  LIN {X -16169.500,Y -1557.401,Z 8.000,A 90.00000,B 0.00000,C 180.00000} ; retreat
  ; Step 222, bar 3419
  LIN {X 16169.500,Y -1557.401,Z 792.630,A 90.00000,B 0.00000,C 180.00000} ; outside
  LIN {X 16169.500,Y -1557.401,Z -42.000,A 90.00000,B 0.00000,C 180.00000} ; preinsert
  LIN {X 16169.500,Y -1557.401,Z -292.000,A 90.00000,B 0.00000,C 180.00000} ; insert
  LIN {X 16169.500,Y -1557.401,Z -292.000,A 90.00000,B 0.00000,C 180.00000} ; release
  LIN {X 16169.500,Y -1557.401,Z 8.000,A 90.00000,B 0.00000,C 180.00000} ; retreat
  ; Step 223, bar 3421
  LIN {X -16169.500,Y 1557.401,Z 792.630,A -90.00000,B 0.00000,C 180.00000} ; outside
  LIN {X -16169.500,Y 1557.401,Z -42.000,A -90.00000,B 0.00000,C 180.00000} ; preinsert
  LIN {X -16169.500,Y 1557.401,Z -292.000,A -90.00000,B 0.00000,C 180.00000} ; insert
  LIN {X -16169.500,Y 1557.401,Z -292.000,A -90.00000,B 0.00000,C 180.00000} ; release
  LIN {X -16169.500,Y 1557.401,Z 8.000,A -90.00000,B 0.00000,C 180.00000} ; retreat
  ; Step 224, bar 3417
  LIN {X 16169.500,Y 1557.401,Z 792.630,A -90.00000,B 0.00000,C 180.00000} ; outside
  LIN {X 16169.500,Y 1557.401,Z -42.000,A -90.00000,B 0.00000,C 180.00000} ; preinsert
  LIN {X 16169.500,Y 1557.401,Z -292.000,A -90.00000,B 0.00000,C 180.00000} ; insert
  LIN {X 16169.500,Y 1557.401,Z -292.000,A -90.00000,B 0.00000,C 180.00000} ; release
  LIN {X 16169.500,Y 1557.401,Z 8.000,A -90.00000,B 0.00000,C 180.00000} ; retreat
  ; Step 225, bar 1865
  LIN {X 0.000,Y -2739.855,Z 792.630,A 0.00000,B 0.00000,C 180.00000} ; outside
  LIN {X 0.000,Y -2739.855,Z -37.029,A 0.00000,B 0.00000,C 180.00000} ; preinsert
  LIN {X 0.000,Y -2739.855,Z -287.029,A 0.00000,B 0.00000,C 180.00000} ; insert
  LIN {X 0.000,Y -2739.855,Z -287.029,A 0.00000,B 0.00000,C 180.00000} ; release
  LIN {X 0.000,Y -2739.855,Z 12.971,A 0.00000,B 0.00000,C 180.00000} ; retreat
  ; Step 226, bar 1878
  LIN {X 0.000,Y 2739.855,Z 792.630,A 0.00000,B 0.00000,C 180.00000} ; outside
  LIN {X 0.000,Y 2739.855,Z -37.029,A 0.00000,B 0.00000,C 180.00000} ; preinsert
  LIN {X 0.000,Y 2739.855,Z -287.029,A 0.00000,B 0.00000,C 180.00000} ; insert
  LIN {X 0.000,Y 2739.855,Z -287.029,A 0.00000,B 0.00000,C 180.00000} ; release
  LIN {X 0.000,Y 2739.855,Z 12.971,A 0.00000,B 0.00000,C 180.00000} ; retreat
  ; Step 227, bar 1060
  LIN {X 16149.984,Y 0.199,Z 793.369,A 90.00387,B 0.00000,C 180.00000} ; outside
  LIN {X 16149.984,Y 0.199,Z -166.684,A 90.00387,B 0.00000,C 180.00000} ; preinsert
  LIN {X 16149.984,Y 0.199,Z -416.684,A 90.00387,B 0.00000,C 180.00000} ; insert
  LIN {X 16149.984,Y 0.199,Z -416.684,A 90.00387,B 0.00000,C 180.00000} ; release
  LIN {X 16149.984,Y 0.199,Z -116.684,A 90.00387,B 0.00000,C 180.00000} ; retreat
  ; Step 228, bar 1061
  LIN {X 16249.984,Y 0.199,Z 793.369,A 90.00387,B 0.00000,C 180.00000} ; outside
  LIN {X 16249.984,Y 0.199,Z -166.684,A 90.00387,B 0.00000,C 180.00000} ; preinsert
  LIN {X 16249.984,Y 0.199,Z -416.684,A 90.00387,B 0.00000,C 180.00000} ; insert
  LIN {X 16249.984,Y 0.199,Z -416.684,A 90.00387,B 0.00000,C 180.00000} ; release
  LIN {X 16249.984,Y 0.199,Z -116.684,A 90.00387,B 0.00000,C 180.00000} ; retreat
  ; Step 229, bar 1847
  LIN {X -16149.984,Y 0.199,Z 793.369,A 89.99613,B 0.00000,C -180.00000} ; outside
  LIN {X -16149.984,Y 0.199,Z -166.684,A 89.99613,B 0.00000,C -180.00000} ; preinsert
  LIN {X -16149.984,Y 0.199,Z -416.684,A 89.99613,B 0.00000,C -180.00000} ; insert
  LIN {X -16149.984,Y 0.199,Z -416.684,A 89.99613,B 0.00000,C -180.00000} ; release
  LIN {X -16149.984,Y 0.199,Z -116.684,A 89.99613,B 0.00000,C -180.00000} ; retreat
  ; Step 230, bar 1848
  LIN {X -16249.984,Y 0.199,Z 793.369,A 89.99613,B 0.00000,C -180.00000} ; outside
  LIN {X -16249.984,Y 0.199,Z -166.684,A 89.99613,B 0.00000,C -180.00000} ; preinsert
  LIN {X -16249.984,Y 0.199,Z -416.684,A 89.99613,B 0.00000,C -180.00000} ; insert
  LIN {X -16249.984,Y 0.199,Z -416.684,A 89.99613,B 0.00000,C -180.00000} ; release
  LIN {X -16249.984,Y 0.199,Z -116.684,A 89.99613,B 0.00000,C -180.00000} ; retreat
  ; Step 231, bar 1051
  LIN {X 15249.971,Y 0.435,Z 793.207,A 89.99774,B 0.00000,C 180.00000} ; outside
  LIN {X 15249.971,Y 0.435,Z -166.823,A 89.99774,B 0.00000,C 180.00000} ; preinsert
  LIN {X 15249.971,Y 0.435,Z -416.823,A 89.99774,B 0.00000,C 180.00000} ; insert
  LIN {X 15249.971,Y 0.435,Z -416.823,A 89.99774,B 0.00000,C 180.00000} ; release
  LIN {X 15249.971,Y 0.435,Z -116.823,A 89.99774,B 0.00000,C 180.00000} ; retreat
  ; Step 232, bar 1052
  LIN {X 15349.971,Y 0.435,Z 793.207,A 89.99774,B 0.00000,C 180.00000} ; outside
  LIN {X 15349.971,Y 0.435,Z -166.823,A 89.99774,B 0.00000,C 180.00000} ; preinsert
  LIN {X 15349.971,Y 0.435,Z -416.823,A 89.99774,B 0.00000,C 180.00000} ; insert
  LIN {X 15349.971,Y 0.435,Z -416.823,A 89.99774,B 0.00000,C 180.00000} ; release
  LIN {X 15349.971,Y 0.435,Z -116.823,A 89.99774,B 0.00000,C 180.00000} ; retreat
  ; Step 233, bar 1053
  LIN {X 15449.971,Y 0.435,Z 793.207,A 89.99774,B 0.00000,C 180.00000} ; outside
  LIN {X 15449.971,Y 0.435,Z -166.823,A 89.99774,B 0.00000,C 180.00000} ; preinsert
  LIN {X 15449.971,Y 0.435,Z -416.823,A 89.99774,B 0.00000,C 180.00000} ; insert
  LIN {X 15449.971,Y 0.435,Z -416.823,A 89.99774,B 0.00000,C 180.00000} ; release
  LIN {X 15449.971,Y 0.435,Z -116.823,A 89.99774,B 0.00000,C 180.00000} ; retreat
  ; Step 234, bar 1055
  LIN {X 15649.971,Y 0.435,Z 793.207,A 89.99774,B 0.00000,C 180.00000} ; outside
  LIN {X 15649.971,Y 0.435,Z -166.823,A 89.99774,B 0.00000,C 180.00000} ; preinsert
  LIN {X 15649.971,Y 0.435,Z -416.823,A 89.99774,B 0.00000,C 180.00000} ; insert
  LIN {X 15649.971,Y 0.435,Z -416.823,A 89.99774,B 0.00000,C 180.00000} ; release
  LIN {X 15649.971,Y 0.435,Z -116.823,A 89.99774,B 0.00000,C 180.00000} ; retreat
  ; Step 235, bar 1056
  LIN {X 15749.971,Y 0.435,Z 793.207,A 89.99774,B 0.00000,C 180.00000} ; outside
  LIN {X 15749.971,Y 0.435,Z -166.823,A 89.99774,B 0.00000,C 180.00000} ; preinsert
  LIN {X 15749.971,Y 0.435,Z -416.823,A 89.99774,B 0.00000,C 180.00000} ; insert
  LIN {X 15749.971,Y 0.435,Z -416.823,A 89.99774,B 0.00000,C 180.00000} ; release
  LIN {X 15749.971,Y 0.435,Z -116.823,A 89.99774,B 0.00000,C 180.00000} ; retreat
  ; Step 236, bar 1057
  LIN {X 15849.971,Y 0.435,Z 793.207,A 89.99774,B 0.00000,C 180.00000} ; outside
  LIN {X 15849.971,Y 0.435,Z -166.823,A 89.99774,B 0.00000,C 180.00000} ; preinsert
  LIN {X 15849.971,Y 0.435,Z -416.823,A 89.99774,B 0.00000,C 180.00000} ; insert
  LIN {X 15849.971,Y 0.435,Z -416.823,A 89.99774,B 0.00000,C 180.00000} ; release
  LIN {X 15849.971,Y 0.435,Z -116.823,A 89.99774,B 0.00000,C 180.00000} ; retreat
  ; Step 237, bar 1058
  LIN {X 15949.971,Y 0.435,Z 793.207,A 89.99774,B 0.00000,C 180.00000} ; outside
  LIN {X 15949.971,Y 0.435,Z -166.823,A 89.99774,B 0.00000,C 180.00000} ; preinsert
  LIN {X 15949.971,Y 0.435,Z -416.823,A 89.99774,B 0.00000,C 180.00000} ; insert
  LIN {X 15949.971,Y 0.435,Z -416.823,A 89.99774,B 0.00000,C 180.00000} ; release
  LIN {X 15949.971,Y 0.435,Z -116.823,A 89.99774,B 0.00000,C 180.00000} ; retreat
  ; Step 238, bar 1059
  LIN {X 16049.971,Y 0.435,Z 793.207,A 89.99774,B 0.00000,C 180.00000} ; outside
  LIN {X 16049.971,Y 0.435,Z -166.823,A 89.99774,B 0.00000,C 180.00000} ; preinsert
  LIN {X 16049.971,Y 0.435,Z -416.823,A 89.99774,B 0.00000,C 180.00000} ; insert
  LIN {X 16049.971,Y 0.435,Z -416.823,A 89.99774,B 0.00000,C 180.00000} ; release
  LIN {X 16049.971,Y 0.435,Z -116.823,A 89.99774,B 0.00000,C 180.00000} ; retreat
  ; Step 239, bar 1799
  LIN {X -15249.971,Y 0.435,Z 793.207,A 90.00226,B 0.00000,C 180.00000} ; outside
  LIN {X -15249.971,Y 0.435,Z -166.823,A 90.00226,B 0.00000,C 180.00000} ; preinsert
  LIN {X -15249.971,Y 0.435,Z -416.823,A 90.00226,B 0.00000,C 180.00000} ; insert
  LIN {X -15249.971,Y 0.435,Z -416.823,A 90.00226,B 0.00000,C 180.00000} ; release
  LIN {X -15249.971,Y 0.435,Z -116.823,A 90.00226,B 0.00000,C 180.00000} ; retreat
  ; Step 240, bar 1800
  LIN {X -15349.971,Y 0.435,Z 793.207,A 90.00226,B 0.00000,C 180.00000} ; outside
  LIN {X -15349.971,Y 0.435,Z -166.823,A 90.00226,B 0.00000,C 180.00000} ; preinsert
  LIN {X -15349.971,Y 0.435,Z -416.823,A 90.00226,B 0.00000,C 180.00000} ; insert
  LIN {X -15349.971,Y 0.435,Z -416.823,A 90.00226,B 0.00000,C 180.00000} ; release
  LIN {X -15349.971,Y 0.435,Z -116.823,A 90.00226,B 0.00000,C 180.00000} ; retreat
  ; Step 241, bar 1801
  LIN {X -15449.971,Y 0.435,Z 793.207,A 90.00226,B 0.00000,C 180.00000} ; outside
  LIN {X -15449.971,Y 0.435,Z -166.823,A 90.00226,B 0.00000,C 180.00000} ; preinsert
  LIN {X -15449.971,Y 0.435,Z -416.823,A 90.00226,B 0.00000,C 180.00000} ; insert
  LIN {X -15449.971,Y 0.435,Z -416.823,A 90.00226,B 0.00000,C 180.00000} ; release
  LIN {X -15449.971,Y 0.435,Z -116.823,A 90.00226,B 0.00000,C 180.00000} ; retreat
  ; Step 242, bar 1802
  LIN {X -15649.971,Y 0.435,Z 793.207,A 90.00226,B 0.00000,C 180.00000} ; outside
  LIN {X -15649.971,Y 0.435,Z -166.823,A 90.00226,B 0.00000,C 180.00000} ; preinsert
  LIN {X -15649.971,Y 0.435,Z -416.823,A 90.00226,B 0.00000,C 180.00000} ; insert
  LIN {X -15649.971,Y 0.435,Z -416.823,A 90.00226,B 0.00000,C 180.00000} ; release
  LIN {X -15649.971,Y 0.435,Z -116.823,A 90.00226,B 0.00000,C 180.00000} ; retreat
  ; Step 243, bar 1803
  LIN {X -15749.971,Y 0.435,Z 793.207,A 90.00226,B 0.00000,C 180.00000} ; outside
  LIN {X -15749.971,Y 0.435,Z -166.823,A 90.00226,B 0.00000,C 180.00000} ; preinsert
  LIN {X -15749.971,Y 0.435,Z -416.823,A 90.00226,B 0.00000,C 180.00000} ; insert
  LIN {X -15749.971,Y 0.435,Z -416.823,A 90.00226,B 0.00000,C 180.00000} ; release
  LIN {X -15749.971,Y 0.435,Z -116.823,A 90.00226,B 0.00000,C 180.00000} ; retreat
  ; Step 244, bar 1804
  LIN {X -15849.971,Y 0.435,Z 793.207,A 90.00226,B 0.00000,C 180.00000} ; outside
  LIN {X -15849.971,Y 0.435,Z -166.823,A 90.00226,B 0.00000,C 180.00000} ; preinsert
  LIN {X -15849.971,Y 0.435,Z -416.823,A 90.00226,B 0.00000,C 180.00000} ; insert
  LIN {X -15849.971,Y 0.435,Z -416.823,A 90.00226,B 0.00000,C 180.00000} ; release
  LIN {X -15849.971,Y 0.435,Z -116.823,A 90.00226,B 0.00000,C 180.00000} ; retreat
  ; Step 245, bar 1805
  LIN {X -15949.971,Y 0.435,Z 793.207,A 90.00226,B 0.00000,C 180.00000} ; outside
  LIN {X -15949.971,Y 0.435,Z -166.823,A 90.00226,B 0.00000,C 180.00000} ; preinsert
  LIN {X -15949.971,Y 0.435,Z -416.823,A 90.00226,B 0.00000,C 180.00000} ; insert
  LIN {X -15949.971,Y 0.435,Z -416.823,A 90.00226,B 0.00000,C 180.00000} ; release
  LIN {X -15949.971,Y 0.435,Z -116.823,A 90.00226,B 0.00000,C 180.00000} ; retreat
  ; Step 246, bar 1806
  LIN {X -16049.971,Y 0.435,Z 793.207,A 90.00226,B 0.00000,C 180.00000} ; outside
  LIN {X -16049.971,Y 0.435,Z -166.823,A 90.00226,B 0.00000,C 180.00000} ; preinsert
  LIN {X -16049.971,Y 0.435,Z -416.823,A 90.00226,B 0.00000,C 180.00000} ; insert
  LIN {X -16049.971,Y 0.435,Z -416.823,A 90.00226,B 0.00000,C 180.00000} ; release
  LIN {X -16049.971,Y 0.435,Z -116.823,A 90.00226,B 0.00000,C 180.00000} ; retreat
  ; Step 247, bar 1866
  LIN {X 0.000,Y -2889.855,Z 792.630,A 0.00000,B 0.00000,C 180.00000} ; outside
  LIN {X 0.000,Y -2889.855,Z -19.788,A 0.00000,B 0.00000,C 180.00000} ; preinsert
  LIN {X 0.000,Y -2889.855,Z -269.788,A 0.00000,B 0.00000,C 180.00000} ; insert
  LIN {X 0.000,Y -2889.855,Z -269.788,A 0.00000,B 0.00000,C 180.00000} ; release
  LIN {X 0.000,Y -2889.855,Z 30.212,A 0.00000,B 0.00000,C 180.00000} ; retreat
  ; Step 248, bar 1879
  LIN {X 0.000,Y 2889.855,Z 792.630,A 0.00000,B 0.00000,C 180.00000} ; outside
  LIN {X 0.000,Y 2889.855,Z -19.788,A 0.00000,B 0.00000,C 180.00000} ; preinsert
  LIN {X 0.000,Y 2889.855,Z -269.788,A 0.00000,B 0.00000,C 180.00000} ; insert
  LIN {X 0.000,Y 2889.855,Z -269.788,A 0.00000,B 0.00000,C 180.00000} ; release
  LIN {X 0.000,Y 2889.855,Z 30.212,A 0.00000,B 0.00000,C 180.00000} ; retreat
  ; Step 249, bar 1050
  LIN {X 15149.971,Y 0.435,Z 793.207,A 89.99774,B 0.00000,C 180.00000} ; outside
  LIN {X 15149.971,Y 0.435,Z -163.267,A 89.99774,B 0.00000,C 180.00000} ; preinsert
  LIN {X 15149.971,Y 0.435,Z -413.267,A 89.99774,B 0.00000,C 180.00000} ; insert
  LIN {X 15149.971,Y 0.435,Z -413.267,A 89.99774,B 0.00000,C 180.00000} ; release
  LIN {X 15149.971,Y 0.435,Z -113.267,A 89.99774,B 0.00000,C 180.00000} ; retreat
  ; Step 250, bar 1798
  LIN {X -15149.971,Y 0.435,Z 793.207,A 90.00226,B 0.00000,C 180.00000} ; outside
  LIN {X -15149.971,Y 0.435,Z -163.267,A 90.00226,B 0.00000,C 180.00000} ; preinsert
  LIN {X -15149.971,Y 0.435,Z -413.267,A 90.00226,B 0.00000,C 180.00000} ; insert
  LIN {X -15149.971,Y 0.435,Z -413.267,A 90.00226,B 0.00000,C 180.00000} ; release
  LIN {X -15149.971,Y 0.435,Z -113.267,A 90.00226,B 0.00000,C 180.00000} ; retreat
  ; Step 251, bar 1049
  LIN {X 15049.971,Y 0.435,Z 793.207,A 89.99774,B 0.00000,C 180.00000} ; outside
  LIN {X 15049.971,Y 0.435,Z -156.587,A 89.99774,B 0.00000,C 180.00000} ; preinsert
  LIN {X 15049.971,Y 0.435,Z -406.587,A 89.99774,B 0.00000,C 180.00000} ; insert
  LIN {X 15049.971,Y 0.435,Z -406.587,A 89.99774,B 0.00000,C 180.00000} ; release
  LIN {X 15049.971,Y 0.435,Z -106.587,A 89.99774,B 0.00000,C 180.00000} ; retreat
  ; Step 252, bar 1797
  LIN {X -15049.971,Y 0.435,Z 793.207,A 90.00226,B 0.00000,C 180.00000} ; outside
  LIN {X -15049.971,Y 0.435,Z -156.587,A 90.00226,B 0.00000,C 180.00000} ; preinsert
  LIN {X -15049.971,Y 0.435,Z -406.587,A 90.00226,B 0.00000,C 180.00000} ; insert
  LIN {X -15049.971,Y 0.435,Z -406.587,A 90.00226,B 0.00000,C 180.00000} ; release
  LIN {X -15049.971,Y 0.435,Z -106.587,A 90.00226,B 0.00000,C 180.00000} ; retreat
  ; Step 253, bar 1048
  LIN {X 14949.971,Y 0.435,Z 793.207,A 89.99774,B 0.00000,C 180.00000} ; outside
  LIN {X 14949.971,Y 0.435,Z -149.906,A 89.99774,B 0.00000,C 180.00000} ; preinsert
  LIN {X 14949.971,Y 0.435,Z -399.906,A 89.99774,B 0.00000,C 180.00000} ; insert
  LIN {X 14949.971,Y 0.435,Z -399.906,A 89.99774,B 0.00000,C 180.00000} ; release
  LIN {X 14949.971,Y 0.435,Z -99.906,A 89.99774,B 0.00000,C 180.00000} ; retreat
  ; Step 254, bar 1796
  LIN {X -14949.971,Y 0.435,Z 793.207,A 90.00226,B 0.00000,C 180.00000} ; outside
  LIN {X -14949.971,Y 0.435,Z -149.906,A 90.00226,B 0.00000,C 180.00000} ; preinsert
  LIN {X -14949.971,Y 0.435,Z -399.906,A 90.00226,B 0.00000,C 180.00000} ; insert
  LIN {X -14949.971,Y 0.435,Z -399.906,A 90.00226,B 0.00000,C 180.00000} ; release
  LIN {X -14949.971,Y 0.435,Z -99.906,A 90.00226,B 0.00000,C 180.00000} ; retreat
  ; Step 255, bar 1950
  LIN {X 0.000,Y -1050.000,Z 792.630,A 0.00000,B 0.00000,C 180.00000} ; outside
  LIN {X 0.000,Y -1050.000,Z -2.875,A 0.00000,B 0.00000,C 180.00000} ; preinsert
  LIN {X 0.000,Y -1050.000,Z -252.875,A 0.00000,B 0.00000,C 180.00000} ; insert
  LIN {X 0.000,Y -1050.000,Z -252.875,A 0.00000,B 0.00000,C 180.00000} ; release
  LIN {X 0.000,Y -1050.000,Z 47.125,A 0.00000,B 0.00000,C 180.00000} ; retreat
  ; Step 256, bar 1945
  LIN {X 0.000,Y 1050.000,Z 792.630,A 0.00000,B 0.00000,C 180.00000} ; outside
  LIN {X 0.000,Y 1050.000,Z -2.875,A 0.00000,B 0.00000,C 180.00000} ; preinsert
  LIN {X 0.000,Y 1050.000,Z -252.875,A 0.00000,B 0.00000,C 180.00000} ; insert
  LIN {X 0.000,Y 1050.000,Z -252.875,A 0.00000,B 0.00000,C 180.00000} ; release
  LIN {X 0.000,Y 1050.000,Z 47.125,A 0.00000,B 0.00000,C 180.00000} ; retreat
  ; Step 257, bar 1867
  LIN {X 0.000,Y -3039.855,Z 792.630,A 0.00000,B 0.00000,C 180.00000} ; outside
  LIN {X 0.000,Y -3039.855,Z -2.546,A 0.00000,B 0.00000,C 180.00000} ; preinsert
  LIN {X 0.000,Y -3039.855,Z -252.546,A 0.00000,B 0.00000,C 180.00000} ; insert
  LIN {X 0.000,Y -3039.855,Z -252.546,A 0.00000,B 0.00000,C 180.00000} ; release
  LIN {X 0.000,Y -3039.855,Z 47.454,A 0.00000,B 0.00000,C 180.00000} ; retreat
  ; Step 258, bar 1880
  LIN {X 0.000,Y 3039.855,Z 792.630,A 0.00000,B 0.00000,C 180.00000} ; outside
  LIN {X 0.000,Y 3039.855,Z -2.546,A 0.00000,B 0.00000,C 180.00000} ; preinsert
  LIN {X 0.000,Y 3039.855,Z -252.546,A 0.00000,B 0.00000,C 180.00000} ; insert
  LIN {X 0.000,Y 3039.855,Z -252.546,A 0.00000,B 0.00000,C 180.00000} ; release
  LIN {X 0.000,Y 3039.855,Z 47.454,A 0.00000,B 0.00000,C 180.00000} ; retreat
  ; Step 259, bar 1047
  LIN {X 14849.971,Y 0.435,Z 793.207,A 89.99774,B 0.00000,C 180.00000} ; outside
  LIN {X 14849.971,Y 0.435,Z -143.225,A 89.99774,B 0.00000,C 180.00000} ; preinsert
  LIN {X 14849.971,Y 0.435,Z -393.225,A 89.99774,B 0.00000,C 180.00000} ; insert
  LIN {X 14849.971,Y 0.435,Z -393.225,A 89.99774,B 0.00000,C 180.00000} ; release
  LIN {X 14849.971,Y 0.435,Z -93.225,A 89.99774,B 0.00000,C 180.00000} ; retreat
  ; Step 260, bar 1795
  LIN {X -14849.971,Y 0.435,Z 793.207,A 90.00226,B 0.00000,C 180.00000} ; outside
  LIN {X -14849.971,Y 0.435,Z -143.225,A 90.00226,B 0.00000,C 180.00000} ; preinsert
  LIN {X -14849.971,Y 0.435,Z -393.225,A 90.00226,B 0.00000,C 180.00000} ; insert
  LIN {X -14849.971,Y 0.435,Z -393.225,A 90.00226,B 0.00000,C 180.00000} ; release
  LIN {X -14849.971,Y 0.435,Z -93.225,A 90.00226,B 0.00000,C 180.00000} ; retreat
  ; Step 261, bar 1046
  LIN {X 14749.971,Y 0.435,Z 793.207,A 89.99774,B 0.00000,C 180.00000} ; outside
  LIN {X 14749.971,Y 0.435,Z -136.544,A 89.99774,B 0.00000,C 180.00000} ; preinsert
  LIN {X 14749.971,Y 0.435,Z -386.544,A 89.99774,B 0.00000,C 180.00000} ; insert
  LIN {X 14749.971,Y 0.435,Z -386.544,A 89.99774,B 0.00000,C 180.00000} ; release
  LIN {X 14749.971,Y 0.435,Z -86.544,A 89.99774,B 0.00000,C 180.00000} ; retreat
  ; Step 262, bar 1794
  LIN {X -14749.971,Y 0.435,Z 793.207,A 90.00226,B 0.00000,C 180.00000} ; outside
  LIN {X -14749.971,Y 0.435,Z -136.544,A 90.00226,B 0.00000,C 180.00000} ; preinsert
  LIN {X -14749.971,Y 0.435,Z -386.544,A 90.00226,B 0.00000,C 180.00000} ; insert
  LIN {X -14749.971,Y 0.435,Z -386.544,A 90.00226,B 0.00000,C 180.00000} ; release
  LIN {X -14749.971,Y 0.435,Z -86.544,A 90.00226,B 0.00000,C 180.00000} ; retreat
  ; Step 263, bar 1868
  LIN {X 0.000,Y -3154.855,Z 792.630,A 0.00000,B 0.00000,C 180.00000} ; outside
  LIN {X 0.000,Y -3154.855,Z 10.672,A 0.00000,B 0.00000,C 180.00000} ; preinsert
  LIN {X 0.000,Y -3154.855,Z -239.328,A 0.00000,B 0.00000,C 180.00000} ; insert
  LIN {X 0.000,Y -3154.855,Z -239.328,A 0.00000,B 0.00000,C 180.00000} ; release
  LIN {X 0.000,Y -3154.855,Z 60.672,A 0.00000,B 0.00000,C 180.00000} ; retreat
  ; Step 264, bar 1881
  LIN {X 0.000,Y 3154.855,Z 792.630,A 0.00000,B 0.00000,C 180.00000} ; outside
  LIN {X 0.000,Y 3154.855,Z 10.672,A 0.00000,B 0.00000,C 180.00000} ; preinsert
  LIN {X 0.000,Y 3154.855,Z -239.328,A 0.00000,B 0.00000,C 180.00000} ; insert
  LIN {X 0.000,Y 3154.855,Z -239.328,A 0.00000,B 0.00000,C 180.00000} ; release
  LIN {X 0.000,Y 3154.855,Z 60.672,A 0.00000,B 0.00000,C 180.00000} ; retreat
  ; Step 265, bar 1045
  LIN {X 14649.971,Y 0.435,Z 793.207,A 89.99774,B 0.00000,C 180.00000} ; outside
  LIN {X 14649.971,Y 0.435,Z -129.863,A 89.99774,B 0.00000,C 180.00000} ; preinsert
  LIN {X 14649.971,Y 0.435,Z -379.863,A 89.99774,B 0.00000,C 180.00000} ; insert
  LIN {X 14649.971,Y 0.435,Z -379.863,A 89.99774,B 0.00000,C 180.00000} ; release
  LIN {X 14649.971,Y 0.435,Z -79.863,A 89.99774,B 0.00000,C 180.00000} ; retreat
  ; Step 266, bar 1793
  LIN {X -14649.971,Y 0.435,Z 793.207,A 90.00226,B 0.00000,C 180.00000} ; outside
  LIN {X -14649.971,Y 0.435,Z -129.863,A 90.00226,B 0.00000,C 180.00000} ; preinsert
  LIN {X -14649.971,Y 0.435,Z -379.863,A 90.00226,B 0.00000,C 180.00000} ; insert
  LIN {X -14649.971,Y 0.435,Z -379.863,A 90.00226,B 0.00000,C 180.00000} ; release
  LIN {X -14649.971,Y 0.435,Z -79.863,A 90.00226,B 0.00000,C 180.00000} ; retreat
  ; Step 267, bar 1869
  LIN {X 0.000,Y -3264.855,Z 798.011,A 0.00000,B 0.00000,C 180.00000} ; outside
  LIN {X 0.000,Y -3264.855,Z 23.316,A 0.00000,B 0.00000,C 180.00000} ; preinsert
  LIN {X 0.000,Y -3264.855,Z -226.684,A 0.00000,B 0.00000,C 180.00000} ; insert
  LIN {X 0.000,Y -3264.855,Z -226.684,A 0.00000,B 0.00000,C 180.00000} ; release
  LIN {X 0.000,Y -3264.855,Z 73.316,A 0.00000,B 0.00000,C 180.00000} ; retreat
  ; Step 268, bar 1882
  LIN {X 0.000,Y 3264.855,Z 798.011,A 0.00000,B 0.00000,C 180.00000} ; outside
  LIN {X 0.000,Y 3264.855,Z 23.316,A 0.00000,B 0.00000,C 180.00000} ; preinsert
  LIN {X 0.000,Y 3264.855,Z -226.684,A 0.00000,B 0.00000,C 180.00000} ; insert
  LIN {X 0.000,Y 3264.855,Z -226.684,A 0.00000,B 0.00000,C 180.00000} ; release
  LIN {X 0.000,Y 3264.855,Z 73.316,A 0.00000,B 0.00000,C 180.00000} ; retreat
  ; Step 269, bar 1043
  LIN {X 14449.971,Y 0.435,Z 793.207,A 89.99774,B 0.00000,C 180.00000} ; outside
  LIN {X 14449.971,Y 0.435,Z -116.502,A 89.99774,B 0.00000,C 180.00000} ; preinsert
  LIN {X 14449.971,Y 0.435,Z -366.502,A 89.99774,B 0.00000,C 180.00000} ; insert
  LIN {X 14449.971,Y 0.435,Z -366.502,A 89.99774,B 0.00000,C 180.00000} ; release
  LIN {X 14449.971,Y 0.435,Z -66.502,A 89.99774,B 0.00000,C 180.00000} ; retreat
  ; Step 270, bar 1792
  LIN {X -14449.971,Y 0.435,Z 793.207,A 90.00226,B 0.00000,C 180.00000} ; outside
  LIN {X -14449.971,Y 0.435,Z -116.502,A 90.00226,B 0.00000,C 180.00000} ; preinsert
  LIN {X -14449.971,Y 0.435,Z -366.502,A 90.00226,B 0.00000,C 180.00000} ; insert
  LIN {X -14449.971,Y 0.435,Z -366.502,A 90.00226,B 0.00000,C 180.00000} ; release
  LIN {X -14449.971,Y 0.435,Z -66.502,A 90.00226,B 0.00000,C 180.00000} ; retreat
  ; Step 271, bar 1870
  LIN {X 0.000,Y -3354.855,Z 818.700,A 0.00000,B 0.00000,C 180.00000} ; outside
  LIN {X 0.000,Y -3354.855,Z 33.661,A 0.00000,B 0.00000,C 180.00000} ; preinsert
  LIN {X 0.000,Y -3354.855,Z -216.339,A 0.00000,B 0.00000,C 180.00000} ; insert
  LIN {X 0.000,Y -3354.855,Z -216.339,A 0.00000,B 0.00000,C 180.00000} ; release
  LIN {X 0.000,Y -3354.855,Z 83.661,A 0.00000,B 0.00000,C 180.00000} ; retreat
  ; Step 272, bar 1883
  LIN {X 0.000,Y 3354.855,Z 818.700,A 0.00000,B 0.00000,C 180.00000} ; outside
  LIN {X 0.000,Y 3354.855,Z 33.661,A 0.00000,B 0.00000,C 180.00000} ; preinsert
  LIN {X 0.000,Y 3354.855,Z -216.339,A 0.00000,B 0.00000,C 180.00000} ; insert
  LIN {X 0.000,Y 3354.855,Z -216.339,A 0.00000,B 0.00000,C 180.00000} ; release
  LIN {X 0.000,Y 3354.855,Z 83.661,A 0.00000,B 0.00000,C 180.00000} ; retreat
  ; Step 273, bar 1042
  LIN {X 14349.971,Y 0.435,Z 793.207,A 89.99774,B 0.00000,C 180.00000} ; outside
  LIN {X 14349.971,Y 0.435,Z -109.821,A 89.99774,B 0.00000,C 180.00000} ; preinsert
  LIN {X 14349.971,Y 0.435,Z -359.821,A 89.99774,B 0.00000,C 180.00000} ; insert
  LIN {X 14349.971,Y 0.435,Z -359.821,A 89.99774,B 0.00000,C 180.00000} ; release
  LIN {X 14349.971,Y 0.435,Z -59.821,A 89.99774,B 0.00000,C 180.00000} ; retreat
  ; Step 274, bar 1791
  LIN {X -14349.971,Y 0.435,Z 793.207,A 90.00226,B 0.00000,C 180.00000} ; outside
  LIN {X -14349.971,Y 0.435,Z -109.821,A 90.00226,B 0.00000,C 180.00000} ; preinsert
  LIN {X -14349.971,Y 0.435,Z -359.821,A 90.00226,B 0.00000,C 180.00000} ; insert
  LIN {X -14349.971,Y 0.435,Z -359.821,A 90.00226,B 0.00000,C 180.00000} ; release
  LIN {X -14349.971,Y 0.435,Z -59.821,A 90.00226,B 0.00000,C 180.00000} ; retreat
  ; Step 275, bar 1041
  LIN {X 14249.971,Y 0.435,Z 793.207,A 89.99774,B 0.00000,C 180.00000} ; outside
  LIN {X 14249.971,Y 0.435,Z -103.140,A 89.99774,B 0.00000,C 180.00000} ; preinsert
  LIN {X 14249.971,Y 0.435,Z -353.140,A 89.99774,B 0.00000,C 180.00000} ; insert
  LIN {X 14249.971,Y 0.435,Z -353.140,A 89.99774,B 0.00000,C 180.00000} ; release
  LIN {X 14249.971,Y 0.435,Z -53.140,A 89.99774,B 0.00000,C 180.00000} ; retreat
  ; Step 276, bar 1790
  LIN {X -14249.971,Y 0.435,Z 793.207,A 90.00226,B 0.00000,C 180.00000} ; outside
  LIN {X -14249.971,Y 0.435,Z -103.140,A 90.00226,B 0.00000,C 180.00000} ; preinsert
  LIN {X -14249.971,Y 0.435,Z -353.140,A 90.00226,B 0.00000,C 180.00000} ; insert
  LIN {X -14249.971,Y 0.435,Z -353.140,A 90.00226,B 0.00000,C 180.00000} ; release
  LIN {X -14249.971,Y 0.435,Z -53.140,A 90.00226,B 0.00000,C 180.00000} ; retreat
  ; Step 277, bar 1040
  LIN {X 14149.971,Y 0.435,Z 793.207,A 89.99774,B 0.00000,C 180.00000} ; outside
  LIN {X 14149.971,Y 0.435,Z -96.459,A 89.99774,B 0.00000,C 180.00000} ; preinsert
  LIN {X 14149.971,Y 0.435,Z -346.459,A 89.99774,B 0.00000,C 180.00000} ; insert
  LIN {X 14149.971,Y 0.435,Z -346.459,A 89.99774,B 0.00000,C 180.00000} ; release
  LIN {X 14149.971,Y 0.435,Z -46.459,A 89.99774,B 0.00000,C 180.00000} ; retreat
  ; Step 278, bar 1789
  LIN {X -14149.971,Y 0.435,Z 793.207,A 90.00226,B 0.00000,C 180.00000} ; outside
  LIN {X -14149.971,Y 0.435,Z -96.459,A 90.00226,B 0.00000,C 180.00000} ; preinsert
  LIN {X -14149.971,Y 0.435,Z -346.459,A 90.00226,B 0.00000,C 180.00000} ; insert
  LIN {X -14149.971,Y 0.435,Z -346.459,A 90.00226,B 0.00000,C 180.00000} ; release
  LIN {X -14149.971,Y 0.435,Z -46.459,A 90.00226,B 0.00000,C 180.00000} ; retreat
  ; Step 279, bar 1944
  LIN {X 0.000,Y -1420.000,Z 849.379,A 0.00000,B 0.00000,C 180.00000} ; outside
  LIN {X 0.000,Y -1420.000,Z 49.000,A 0.00000,B 0.00000,C 180.00000} ; preinsert
  LIN {X 0.000,Y -1420.000,Z -201.000,A 0.00000,B 0.00000,C 180.00000} ; insert
  LIN {X 0.000,Y -1420.000,Z -201.000,A 0.00000,B 0.00000,C 180.00000} ; release
  LIN {X 0.000,Y -1420.000,Z 99.000,A 0.00000,B 0.00000,C 180.00000} ; retreat
  ; Step 280, bar 1943
  LIN {X 0.000,Y -1050.000,Z 849.379,A 0.00000,B 0.00000,C 180.00000} ; outside
  LIN {X 0.000,Y -1050.000,Z 49.000,A 0.00000,B 0.00000,C 180.00000} ; preinsert
  LIN {X 0.000,Y -1050.000,Z -201.000,A 0.00000,B 0.00000,C 180.00000} ; insert
  LIN {X 0.000,Y -1050.000,Z -201.000,A 0.00000,B 0.00000,C 180.00000} ; release
  LIN {X 0.000,Y -1050.000,Z 99.000,A 0.00000,B 0.00000,C 180.00000} ; retreat
  ; Step 281, bar 1942
  LIN {X 0.000,Y -875.000,Z 849.379,A 0.00000,B 0.00000,C 180.00000} ; outside
  LIN {X 0.000,Y -875.000,Z 49.000,A 0.00000,B 0.00000,C 180.00000} ; preinsert
  LIN {X 0.000,Y -875.000,Z -201.000,A 0.00000,B 0.00000,C 180.00000} ; insert
  LIN {X 0.000,Y -875.000,Z -201.000,A 0.00000,B 0.00000,C 180.00000} ; release
  LIN {X 0.000,Y -875.000,Z 99.000,A 0.00000,B 0.00000,C 180.00000} ; retreat
  ; Step 282, bar 1941
  LIN {X 0.000,Y -750.000,Z 849.379,A 0.00000,B 0.00000,C 180.00000} ; outside
  LIN {X 0.000,Y -750.000,Z 49.000,A 0.00000,B 0.00000,C 180.00000} ; preinsert
  LIN {X 0.000,Y -750.000,Z -201.000,A 0.00000,B 0.00000,C 180.00000} ; insert
  LIN {X 0.000,Y -750.000,Z -201.000,A 0.00000,B 0.00000,C 180.00000} ; release
  LIN {X 0.000,Y -750.000,Z 99.000,A 0.00000,B 0.00000,C 180.00000} ; retreat
  ; Step 283, bar 1940
  LIN {X 0.000,Y -625.000,Z 849.379,A 0.00000,B 0.00000,C 180.00000} ; outside
  LIN {X 0.000,Y -625.000,Z 49.000,A 0.00000,B 0.00000,C 180.00000} ; preinsert
  LIN {X 0.000,Y -625.000,Z -201.000,A 0.00000,B 0.00000,C 180.00000} ; insert
  LIN {X 0.000,Y -625.000,Z -201.000,A 0.00000,B 0.00000,C 180.00000} ; release
  LIN {X 0.000,Y -625.000,Z 99.000,A 0.00000,B 0.00000,C 180.00000} ; retreat
  ; Step 284, bar 1939
  LIN {X 0.000,Y -500.000,Z 849.379,A 0.00000,B 0.00000,C 180.00000} ; outside
  LIN {X 0.000,Y -500.000,Z 49.000,A 0.00000,B 0.00000,C 180.00000} ; preinsert
  LIN {X 0.000,Y -500.000,Z -201.000,A 0.00000,B 0.00000,C 180.00000} ; insert
  LIN {X 0.000,Y -500.000,Z -201.000,A 0.00000,B 0.00000,C 180.00000} ; release
  LIN {X 0.000,Y -500.000,Z 99.000,A 0.00000,B 0.00000,C 180.00000} ; retreat
  ; Step 285, bar 1938
  LIN {X 0.000,Y -375.000,Z 849.379,A 0.00000,B 0.00000,C 180.00000} ; outside
  LIN {X 0.000,Y -375.000,Z 49.000,A 0.00000,B 0.00000,C 180.00000} ; preinsert
  LIN {X 0.000,Y -375.000,Z -201.000,A 0.00000,B 0.00000,C 180.00000} ; insert
  LIN {X 0.000,Y -375.000,Z -201.000,A 0.00000,B 0.00000,C 180.00000} ; release
  LIN {X 0.000,Y -375.000,Z 99.000,A 0.00000,B 0.00000,C 180.00000} ; retreat
  ; Step 286, bar 1937
  LIN {X 0.000,Y -250.000,Z 849.379,A 0.00000,B 0.00000,C 180.00000} ; outside
  LIN {X 0.000,Y -250.000,Z 49.000,A 0.00000,B 0.00000,C 180.00000} ; preinsert
  LIN {X 0.000,Y -250.000,Z -201.000,A 0.00000,B 0.00000,C 180.00000} ; insert
  LIN {X 0.000,Y -250.000,Z -201.000,A 0.00000,B 0.00000,C 180.00000} ; release
  LIN {X 0.000,Y -250.000,Z 99.000,A 0.00000,B 0.00000,C 180.00000} ; retreat
  ; Step 287, bar 1936
  LIN {X 0.000,Y -125.000,Z 849.379,A 0.00000,B 0.00000,C 180.00000} ; outside
  LIN {X 0.000,Y -125.000,Z 49.000,A 0.00000,B 0.00000,C 180.00000} ; preinsert
  LIN {X 0.000,Y -125.000,Z -201.000,A 0.00000,B 0.00000,C 180.00000} ; insert
  LIN {X 0.000,Y -125.000,Z -201.000,A 0.00000,B 0.00000,C 180.00000} ; release
  LIN {X 0.000,Y -125.000,Z 99.000,A 0.00000,B 0.00000,C 180.00000} ; retreat
  ; Step 288, bar 893
  LIN {X 0.000,Y 0.000,Z 849.379,A 0.00000,B 0.00000,C 180.00000} ; outside
  LIN {X 0.000,Y 0.000,Z 49.000,A 0.00000,B 0.00000,C 180.00000} ; preinsert
  LIN {X 0.000,Y 0.000,Z -201.000,A 0.00000,B 0.00000,C 180.00000} ; insert
  LIN {X 0.000,Y 0.000,Z -201.000,A 0.00000,B 0.00000,C 180.00000} ; release
  LIN {X 0.000,Y 0.000,Z 99.000,A 0.00000,B 0.00000,C 180.00000} ; retreat
  ; Step 289, bar 1927
  LIN {X 0.000,Y 125.000,Z 849.379,A 0.00000,B 0.00000,C 180.00000} ; outside
  LIN {X 0.000,Y 125.000,Z 49.000,A 0.00000,B 0.00000,C 180.00000} ; preinsert
  LIN {X 0.000,Y 125.000,Z -201.000,A 0.00000,B 0.00000,C 180.00000} ; insert
  LIN {X 0.000,Y 125.000,Z -201.000,A 0.00000,B 0.00000,C 180.00000} ; release
  LIN {X 0.000,Y 125.000,Z 99.000,A 0.00000,B 0.00000,C 180.00000} ; retreat
  ; Step 290, bar 1928
  LIN {X 0.000,Y 250.000,Z 849.379,A 0.00000,B 0.00000,C 180.00000} ; outside
  LIN {X 0.000,Y 250.000,Z 49.000,A 0.00000,B 0.00000,C 180.00000} ; preinsert
  LIN {X 0.000,Y 250.000,Z -201.000,A 0.00000,B 0.00000,C 180.00000} ; insert
  LIN {X 0.000,Y 250.000,Z -201.000,A 0.00000,B 0.00000,C 180.00000} ; release
  LIN {X 0.000,Y 250.000,Z 99.000,A 0.00000,B 0.00000,C 180.00000} ; retreat
  ; Step 291, bar 1929
  LIN {X 0.000,Y 375.000,Z 849.379,A 0.00000,B 0.00000,C 180.00000} ; outside
  LIN {X 0.000,Y 375.000,Z 49.000,A 0.00000,B 0.00000,C 180.00000} ; preinsert
  LIN {X 0.000,Y 375.000,Z -201.000,A 0.00000,B 0.00000,C 180.00000} ; insert
  LIN {X 0.000,Y 375.000,Z -201.000,A 0.00000,B 0.00000,C 180.00000} ; release
  LIN {X 0.000,Y 375.000,Z 99.000,A 0.00000,B 0.00000,C 180.00000} ; retreat
  ; Step 292, bar 1930
  LIN {X 0.000,Y 500.000,Z 849.379,A 0.00000,B 0.00000,C 180.00000} ; outside
  LIN {X 0.000,Y 500.000,Z 49.000,A 0.00000,B 0.00000,C 180.00000} ; preinsert
  LIN {X 0.000,Y 500.000,Z -201.000,A 0.00000,B 0.00000,C 180.00000} ; insert
  LIN {X 0.000,Y 500.000,Z -201.000,A 0.00000,B 0.00000,C 180.00000} ; release
  LIN {X 0.000,Y 500.000,Z 99.000,A 0.00000,B 0.00000,C 180.00000} ; retreat
  ; Step 293, bar 1931
  LIN {X 0.000,Y 625.000,Z 849.379,A 0.00000,B 0.00000,C 180.00000} ; outside
  LIN {X 0.000,Y 625.000,Z 49.000,A 0.00000,B 0.00000,C 180.00000} ; preinsert
  LIN {X 0.000,Y 625.000,Z -201.000,A 0.00000,B 0.00000,C 180.00000} ; insert
  LIN {X 0.000,Y 625.000,Z -201.000,A 0.00000,B 0.00000,C 180.00000} ; release
  LIN {X 0.000,Y 625.000,Z 99.000,A 0.00000,B 0.00000,C 180.00000} ; retreat
  ; Step 294, bar 1932
  LIN {X 0.000,Y 750.000,Z 849.379,A 0.00000,B 0.00000,C 180.00000} ; outside
  LIN {X 0.000,Y 750.000,Z 49.000,A 0.00000,B 0.00000,C 180.00000} ; preinsert
  LIN {X 0.000,Y 750.000,Z -201.000,A 0.00000,B 0.00000,C 180.00000} ; insert
  LIN {X 0.000,Y 750.000,Z -201.000,A 0.00000,B 0.00000,C 180.00000} ; release
  LIN {X 0.000,Y 750.000,Z 99.000,A 0.00000,B 0.00000,C 180.00000} ; retreat
  ; Step 295, bar 1933
  LIN {X 0.000,Y 875.000,Z 849.379,A 0.00000,B 0.00000,C 180.00000} ; outside
  LIN {X 0.000,Y 875.000,Z 49.000,A 0.00000,B 0.00000,C 180.00000} ; preinsert
  LIN {X 0.000,Y 875.000,Z -201.000,A 0.00000,B 0.00000,C 180.00000} ; insert
  LIN {X 0.000,Y 875.000,Z -201.000,A 0.00000,B 0.00000,C 180.00000} ; release
  LIN {X 0.000,Y 875.000,Z 99.000,A 0.00000,B 0.00000,C 180.00000} ; retreat
  ; Step 296, bar 1934
  LIN {X 0.000,Y 1050.000,Z 849.379,A 0.00000,B 0.00000,C 180.00000} ; outside
  LIN {X 0.000,Y 1050.000,Z 49.000,A 0.00000,B 0.00000,C 180.00000} ; preinsert
  LIN {X 0.000,Y 1050.000,Z -201.000,A 0.00000,B 0.00000,C 180.00000} ; insert
  LIN {X 0.000,Y 1050.000,Z -201.000,A 0.00000,B 0.00000,C 180.00000} ; release
  LIN {X 0.000,Y 1050.000,Z 99.000,A 0.00000,B 0.00000,C 180.00000} ; retreat
  ; Step 297, bar 1935
  LIN {X 0.000,Y 1420.000,Z 849.379,A 0.00000,B 0.00000,C 180.00000} ; outside
  LIN {X 0.000,Y 1420.000,Z 49.000,A 0.00000,B 0.00000,C 180.00000} ; preinsert
  LIN {X 0.000,Y 1420.000,Z -201.000,A 0.00000,B 0.00000,C 180.00000} ; insert
  LIN {X 0.000,Y 1420.000,Z -201.000,A 0.00000,B 0.00000,C 180.00000} ; release
  LIN {X 0.000,Y 1420.000,Z 99.000,A 0.00000,B 0.00000,C 180.00000} ; retreat
  ; Step 298, bar 1062
  LIN {X 16149.984,Y 0.199,Z 793.369,A 90.00387,B 0.00000,C 180.00000} ; outside
  LIN {X 16149.984,Y 0.199,Z -91.684,A 90.00387,B 0.00000,C 180.00000} ; preinsert
  LIN {X 16149.984,Y 0.199,Z -341.684,A 90.00387,B 0.00000,C 180.00000} ; insert
  LIN {X 16149.984,Y 0.199,Z -341.684,A 90.00387,B 0.00000,C 180.00000} ; release
  LIN {X 16149.984,Y 0.199,Z -41.684,A 90.00387,B 0.00000,C 180.00000} ; retreat
  ; Step 299, bar 1063
  LIN {X 16249.984,Y 0.199,Z 793.369,A 90.00387,B 0.00000,C 180.00000} ; outside
  LIN {X 16249.984,Y 0.199,Z -91.684,A 90.00387,B 0.00000,C 180.00000} ; preinsert
  LIN {X 16249.984,Y 0.199,Z -341.684,A 90.00387,B 0.00000,C 180.00000} ; insert
  LIN {X 16249.984,Y 0.199,Z -341.684,A 90.00387,B 0.00000,C 180.00000} ; release
  LIN {X 16249.984,Y 0.199,Z -41.684,A 90.00387,B 0.00000,C 180.00000} ; retreat
  ; Step 300, bar 1849
  LIN {X -16149.984,Y 0.199,Z 793.369,A 89.99613,B 0.00000,C -180.00000} ; outside
  LIN {X -16149.984,Y 0.199,Z -91.684,A 89.99613,B 0.00000,C -180.00000} ; preinsert
  LIN {X -16149.984,Y 0.199,Z -341.684,A 89.99613,B 0.00000,C -180.00000} ; insert
  LIN {X -16149.984,Y 0.199,Z -341.684,A 89.99613,B 0.00000,C -180.00000} ; release
  LIN {X -16149.984,Y 0.199,Z -41.684,A 89.99613,B 0.00000,C -180.00000} ; retreat
  ; Step 301, bar 1850
  LIN {X -16249.984,Y 0.199,Z 793.369,A 89.99613,B 0.00000,C -180.00000} ; outside
  LIN {X -16249.984,Y 0.199,Z -91.684,A 89.99613,B 0.00000,C -180.00000} ; preinsert
  LIN {X -16249.984,Y 0.199,Z -341.684,A 89.99613,B 0.00000,C -180.00000} ; insert
  LIN {X -16249.984,Y 0.199,Z -341.684,A 89.99613,B 0.00000,C -180.00000} ; release
  LIN {X -16249.984,Y 0.199,Z -41.684,A 89.99613,B 0.00000,C -180.00000} ; retreat
  ; Step 302, bar 1871
  LIN {X 0.000,Y -3489.855,Z 858.485,A 0.00000,B 0.00000,C 180.00000} ; outside
  LIN {X 0.000,Y -3489.855,Z 53.553,A 0.00000,B 0.00000,C 180.00000} ; preinsert
  LIN {X 0.000,Y -3489.855,Z -196.447,A 0.00000,B 0.00000,C 180.00000} ; insert
  LIN {X 0.000,Y -3489.855,Z -196.447,A 0.00000,B 0.00000,C 180.00000} ; release
  LIN {X 0.000,Y -3489.855,Z 103.553,A 0.00000,B 0.00000,C 180.00000} ; retreat
  ; Step 303, bar 1884
  LIN {X 0.000,Y 3489.855,Z 858.485,A 0.00000,B 0.00000,C 180.00000} ; outside
  LIN {X 0.000,Y 3489.855,Z 53.553,A 0.00000,B 0.00000,C 180.00000} ; preinsert
  LIN {X 0.000,Y 3489.855,Z -196.447,A 0.00000,B 0.00000,C 180.00000} ; insert
  LIN {X 0.000,Y 3489.855,Z -196.447,A 0.00000,B 0.00000,C 180.00000} ; release
  LIN {X 0.000,Y 3489.855,Z 103.553,A 0.00000,B 0.00000,C 180.00000} ; retreat
  ; Step 304, bar 1039
  LIN {X 14049.971,Y 0.435,Z 793.207,A 89.99774,B 0.00000,C 180.00000} ; outside
  LIN {X 14049.971,Y 0.435,Z -89.778,A 89.99774,B 0.00000,C 180.00000} ; preinsert
  LIN {X 14049.971,Y 0.435,Z -339.778,A 89.99774,B 0.00000,C 180.00000} ; insert
  LIN {X 14049.971,Y 0.435,Z -339.778,A 89.99774,B 0.00000,C 180.00000} ; release
  LIN {X 14049.971,Y 0.435,Z -39.778,A 89.99774,B 0.00000,C 180.00000} ; retreat
  ; Step 305, bar 1788
  LIN {X -14049.971,Y 0.435,Z 793.207,A 90.00226,B 0.00000,C 180.00000} ; outside
  LIN {X -14049.971,Y 0.435,Z -89.778,A 90.00226,B 0.00000,C 180.00000} ; preinsert
  LIN {X -14049.971,Y 0.435,Z -339.778,A 90.00226,B 0.00000,C 180.00000} ; insert
  LIN {X -14049.971,Y 0.435,Z -339.778,A 90.00226,B 0.00000,C 180.00000} ; release
  LIN {X -14049.971,Y 0.435,Z -39.778,A 90.00226,B 0.00000,C 180.00000} ; retreat
  ; Step 306, bar 1038
  LIN {X 13949.971,Y 0.435,Z 793.207,A 89.99774,B 0.00000,C 180.00000} ; outside
  LIN {X 13949.971,Y 0.435,Z -83.097,A 89.99774,B 0.00000,C 180.00000} ; preinsert
  LIN {X 13949.971,Y 0.435,Z -333.097,A 89.99774,B 0.00000,C 180.00000} ; insert
  LIN {X 13949.971,Y 0.435,Z -333.097,A 89.99774,B 0.00000,C 180.00000} ; release
  LIN {X 13949.971,Y 0.435,Z -33.097,A 89.99774,B 0.00000,C 180.00000} ; retreat
  ; Step 307, bar 1787
  LIN {X -13949.971,Y 0.435,Z 793.207,A 90.00226,B 0.00000,C 180.00000} ; outside
  LIN {X -13949.971,Y 0.435,Z -83.097,A 90.00226,B 0.00000,C 180.00000} ; preinsert
  LIN {X -13949.971,Y 0.435,Z -333.097,A 90.00226,B 0.00000,C 180.00000} ; insert
  LIN {X -13949.971,Y 0.435,Z -333.097,A 90.00226,B 0.00000,C 180.00000} ; release
  LIN {X -13949.971,Y 0.435,Z -33.097,A 90.00226,B 0.00000,C 180.00000} ; retreat
  ; Step 308, bar 1250
  LIN {X -13665.921,Y 0.110,Z 792.800,A 89.99666,B 0.00000,C 180.00000} ; outside
  LIN {X -13665.921,Y 0.110,Z -63.076,A 89.99666,B 0.00000,C 180.00000} ; preinsert
  LIN {X -13665.921,Y 0.110,Z -313.076,A 89.99666,B 0.00000,C 180.00000} ; insert
  LIN {X -13665.921,Y 0.110,Z -313.076,A 89.99666,B 0.00000,C 180.00000} ; release
  LIN {X -13665.921,Y 0.110,Z -13.076,A 89.99666,B 0.00000,C 180.00000} ; retreat
  ; Step 309, bar 1246
  LIN {X -13649.921,Y 0.110,Z 792.800,A 89.99666,B 0.00000,C 180.00000} ; outside
  LIN {X -13649.921,Y 0.110,Z -63.076,A 89.99666,B 0.00000,C 180.00000} ; preinsert
  LIN {X -13649.921,Y 0.110,Z -313.076,A 89.99666,B 0.00000,C 180.00000} ; insert
  LIN {X -13649.921,Y 0.110,Z -313.076,A 89.99666,B 0.00000,C 180.00000} ; release
  LIN {X -13649.921,Y 0.110,Z -13.076,A 89.99666,B 0.00000,C 180.00000} ; retreat
  ; Step 310, bar 1031
  LIN {X 13649.921,Y 0.097,Z 792.800,A 90.00334,B 0.00000,C 180.00000} ; outside
  LIN {X 13649.921,Y 0.097,Z -63.076,A 90.00334,B 0.00000,C 180.00000} ; preinsert
  LIN {X 13649.921,Y 0.097,Z -313.076,A 90.00334,B 0.00000,C 180.00000} ; insert
  LIN {X 13649.921,Y 0.097,Z -313.076,A 90.00334,B 0.00000,C 180.00000} ; release
  LIN {X 13649.921,Y 0.097,Z -13.076,A 90.00334,B 0.00000,C 180.00000} ; retreat
  ; Step 311, bar 1036
  LIN {X 13665.921,Y 0.097,Z 792.800,A 90.00334,B 0.00000,C 180.00000} ; outside
  LIN {X 13665.921,Y 0.097,Z -63.076,A 90.00334,B 0.00000,C 180.00000} ; preinsert
  LIN {X 13665.921,Y 0.097,Z -313.076,A 90.00334,B 0.00000,C 180.00000} ; insert
  LIN {X 13665.921,Y 0.097,Z -313.076,A 90.00334,B 0.00000,C 180.00000} ; release
  LIN {X 13665.921,Y 0.097,Z -13.076,A 90.00334,B 0.00000,C 180.00000} ; retreat
  ; Step 312, bar 1037
  LIN {X 13849.971,Y 0.435,Z 793.207,A 89.99774,B 0.00000,C 180.00000} ; outside
  LIN {X 13849.971,Y 0.435,Z -76.416,A 89.99774,B 0.00000,C 180.00000} ; preinsert
  LIN {X 13849.971,Y 0.435,Z -326.416,A 89.99774,B 0.00000,C 180.00000} ; insert
  LIN {X 13849.971,Y 0.435,Z -326.416,A 89.99774,B 0.00000,C 180.00000} ; release
  LIN {X 13849.971,Y 0.435,Z -26.416,A 89.99774,B 0.00000,C 180.00000} ; retreat
  ; Step 313, bar 1786
  LIN {X -13849.971,Y 0.435,Z 793.207,A 90.00226,B 0.00000,C 180.00000} ; outside
  LIN {X -13849.971,Y 0.435,Z -76.416,A 90.00226,B 0.00000,C 180.00000} ; preinsert
  LIN {X -13849.971,Y 0.435,Z -326.416,A 90.00226,B 0.00000,C 180.00000} ; insert
  LIN {X -13849.971,Y 0.435,Z -326.416,A 90.00226,B 0.00000,C 180.00000} ; release
  LIN {X -13849.971,Y 0.435,Z -26.416,A 90.00226,B 0.00000,C 180.00000} ; retreat
  ; Step 314, bar 1245
  LIN {X -13549.921,Y 0.110,Z 792.800,A 89.99666,B 0.00000,C 180.00000} ; outside
  LIN {X -13549.921,Y 0.110,Z -56.395,A 89.99666,B 0.00000,C 180.00000} ; preinsert
  LIN {X -13549.921,Y 0.110,Z -306.395,A 89.99666,B 0.00000,C 180.00000} ; insert
  LIN {X -13549.921,Y 0.110,Z -306.395,A 89.99666,B 0.00000,C 180.00000} ; release
  LIN {X -13549.921,Y 0.110,Z -6.395,A 89.99666,B 0.00000,C 180.00000} ; retreat
  ; Step 315, bar 1030
  LIN {X 13549.921,Y 0.097,Z 792.800,A 90.00334,B 0.00000,C 180.00000} ; outside
  LIN {X 13549.921,Y 0.097,Z -56.395,A 90.00334,B 0.00000,C 180.00000} ; preinsert
  LIN {X 13549.921,Y 0.097,Z -306.395,A 90.00334,B 0.00000,C 180.00000} ; insert
  LIN {X 13549.921,Y 0.097,Z -306.395,A 90.00334,B 0.00000,C 180.00000} ; release
  LIN {X 13549.921,Y 0.097,Z -6.395,A 90.00334,B 0.00000,C 180.00000} ; retreat
  ; Step 316, bar 1032
  LIN {X 13749.971,Y 0.435,Z 793.207,A 89.99774,B 0.00000,C 180.00000} ; outside
  LIN {X 13749.971,Y 0.435,Z -69.736,A 89.99774,B 0.00000,C 180.00000} ; preinsert
  LIN {X 13749.971,Y 0.435,Z -319.736,A 89.99774,B 0.00000,C 180.00000} ; insert
  LIN {X 13749.971,Y 0.435,Z -319.736,A 89.99774,B 0.00000,C 180.00000} ; release
  LIN {X 13749.971,Y 0.435,Z -19.736,A 89.99774,B 0.00000,C 180.00000} ; retreat
  ; Step 317, bar 1785
  LIN {X -13749.971,Y 0.435,Z 793.207,A 90.00226,B 0.00000,C 180.00000} ; outside
  LIN {X -13749.971,Y 0.435,Z -69.736,A 90.00226,B 0.00000,C 180.00000} ; preinsert
  LIN {X -13749.971,Y 0.435,Z -319.736,A 90.00226,B 0.00000,C 180.00000} ; insert
  LIN {X -13749.971,Y 0.435,Z -319.736,A 90.00226,B 0.00000,C 180.00000} ; release
  LIN {X -13749.971,Y 0.435,Z -19.736,A 90.00226,B 0.00000,C 180.00000} ; retreat
  ; Step 318, bar 1244
  LIN {X -13449.921,Y 0.110,Z 792.800,A 89.99666,B 0.00000,C 180.00000} ; outside
  LIN {X -13449.921,Y 0.110,Z -49.714,A 89.99666,B 0.00000,C 180.00000} ; preinsert
  LIN {X -13449.921,Y 0.110,Z -299.714,A 89.99666,B 0.00000,C 180.00000} ; insert
  LIN {X -13449.921,Y 0.110,Z -299.714,A 89.99666,B 0.00000,C 180.00000} ; release
  LIN {X -13449.921,Y 0.110,Z 0.286,A 89.99666,B 0.00000,C 180.00000} ; retreat
  ; Step 319, bar 1029
  LIN {X 13449.921,Y 0.097,Z 792.800,A 90.00334,B 0.00000,C 180.00000} ; outside
  LIN {X 13449.921,Y 0.097,Z -49.714,A 90.00334,B 0.00000,C 180.00000} ; preinsert
  LIN {X 13449.921,Y 0.097,Z -299.714,A 90.00334,B 0.00000,C 180.00000} ; insert
  LIN {X 13449.921,Y 0.097,Z -299.714,A 90.00334,B 0.00000,C 180.00000} ; release
  LIN {X 13449.921,Y 0.097,Z 0.286,A 90.00334,B 0.00000,C 180.00000} ; retreat
  ; Step 320, bar 3293
  LIN {X -15485.187,Y -1114.878,Z 914.125,A -134.96824,B 0.00000,C -180.00000} ; outside
  LIN {X -15485.187,Y -1114.878,Z 81.232,A -134.96824,B 0.00000,C -180.00000} ; preinsert
  LIN {X -15485.187,Y -1114.878,Z -168.768,A -134.96824,B 0.00000,C -180.00000} ; insert
  LIN {X -15485.187,Y -1114.878,Z -168.768,A -134.96824,B 0.00000,C -180.00000} ; release
  LIN {X -15485.187,Y -1114.878,Z 131.232,A -134.96824,B 0.00000,C -180.00000} ; retreat
  ; Step 321, bar 3295
  LIN {X -15614.813,Y -1114.878,Z 914.288,A -45.03176,B 0.00000,C 180.00000} ; outside
  LIN {X -15614.813,Y -1114.878,Z 81.232,A -45.03176,B 0.00000,C 180.00000} ; preinsert
  LIN {X -15614.813,Y -1114.878,Z -168.768,A -45.03176,B 0.00000,C 180.00000} ; insert
  LIN {X -15614.813,Y -1114.878,Z -168.768,A -45.03176,B 0.00000,C 180.00000} ; release
  LIN {X -15614.813,Y -1114.878,Z 131.232,A -45.03176,B 0.00000,C 180.00000} ; retreat
  ; Step 322, bar 3373
  LIN {X 15485.187,Y -1114.878,Z 914.288,A -45.03176,B 0.00000,C 180.00000} ; outside
  LIN {X 15485.187,Y -1114.878,Z 81.232,A -45.03176,B 0.00000,C 180.00000} ; preinsert
  LIN {X 15485.187,Y -1114.878,Z -168.768,A -45.03176,B 0.00000,C 180.00000} ; insert
  LIN {X 15485.187,Y -1114.878,Z -168.768,A -45.03176,B 0.00000,C 180.00000} ; release
  LIN {X 15485.187,Y -1114.878,Z 131.232,A -45.03176,B 0.00000,C 180.00000} ; retreat
  ; Step 323, bar 3375
  LIN {X 15614.813,Y -1114.878,Z 914.125,A -134.96824,B 0.00000,C -180.00000} ; outside
  LIN {X 15614.813,Y -1114.878,Z 81.232,A -134.96824,B 0.00000,C -180.00000} ; preinsert
  LIN {X 15614.813,Y -1114.878,Z -168.768,A -134.96824,B 0.00000,C -180.00000} ; insert
  LIN {X 15614.813,Y -1114.878,Z -168.768,A -134.96824,B 0.00000,C -180.00000} ; release
  LIN {X 15614.813,Y -1114.878,Z 131.232,A -134.96824,B 0.00000,C -180.00000} ; retreat
  ; Step 324, bar 3294
  LIN {X -15485.122,Y -985.187,Z 914.125,A -44.96824,B 0.00000,C 180.00000} ; outside
  LIN {X -15485.122,Y -985.187,Z 81.232,A -44.96824,B 0.00000,C 180.00000} ; preinsert
  LIN {X -15485.122,Y -985.187,Z -168.768,A -44.96824,B 0.00000,C 180.00000} ; insert
  LIN {X -15485.122,Y -985.187,Z -168.768,A -44.96824,B 0.00000,C 180.00000} ; release
  LIN {X -15485.122,Y -985.187,Z 131.232,A -44.96824,B 0.00000,C 180.00000} ; retreat
  ; Step 325, bar 3292
  LIN {X -15614.878,Y -985.187,Z 914.288,A -135.03176,B 0.00000,C -180.00000} ; outside
  LIN {X -15614.878,Y -985.187,Z 81.232,A -135.03176,B 0.00000,C -180.00000} ; preinsert
  LIN {X -15614.878,Y -985.187,Z -168.768,A -135.03176,B 0.00000,C -180.00000} ; insert
  LIN {X -15614.878,Y -985.187,Z -168.768,A -135.03176,B 0.00000,C -180.00000} ; release
  LIN {X -15614.878,Y -985.187,Z 131.232,A -135.03176,B 0.00000,C -180.00000} ; retreat
  ; Step 326, bar 3374
  LIN {X 15485.122,Y -985.187,Z 914.288,A -135.03176,B 0.00000,C 180.00000} ; outside
  LIN {X 15485.122,Y -985.187,Z 81.232,A -135.03176,B 0.00000,C 180.00000} ; preinsert
  LIN {X 15485.122,Y -985.187,Z -168.768,A -135.03176,B 0.00000,C 180.00000} ; insert
  LIN {X 15485.122,Y -985.187,Z -168.768,A -135.03176,B 0.00000,C 180.00000} ; release
  LIN {X 15485.122,Y -985.187,Z 131.232,A -135.03176,B 0.00000,C 180.00000} ; retreat
  ; Step 327, bar 3372
  LIN {X 15614.878,Y -985.187,Z 914.125,A -44.96824,B 0.00000,C 180.00000} ; outside
  LIN {X 15614.878,Y -985.187,Z 81.232,A -44.96824,B 0.00000,C 180.00000} ; preinsert
  LIN {X 15614.878,Y -985.187,Z -168.768,A -44.96824,B 0.00000,C 180.00000} ; insert
  LIN {X 15614.878,Y -985.187,Z -168.768,A -44.96824,B 0.00000,C 180.00000} ; release
  LIN {X 15614.878,Y -985.187,Z 131.232,A -44.96824,B 0.00000,C 180.00000} ; retreat
  ; Step 328, bar 3332
  LIN {X -15614.878,Y 985.187,Z 914.125,A 135.03176,B 0.00000,C 180.00000} ; outside
  LIN {X -15614.878,Y 985.187,Z 81.232,A 135.03176,B 0.00000,C 180.00000} ; preinsert
  LIN {X -15614.878,Y 985.187,Z -168.768,A 135.03176,B 0.00000,C 180.00000} ; insert
  LIN {X -15614.878,Y 985.187,Z -168.768,A 135.03176,B 0.00000,C 180.00000} ; release
  LIN {X -15614.878,Y 985.187,Z 131.232,A 135.03176,B 0.00000,C 180.00000} ; retreat
  ; Step 329, bar 3412
  LIN {X 15614.878,Y 985.187,Z 914.288,A 44.96824,B 0.00000,C 180.00000} ; outside
  LIN {X 15614.878,Y 985.187,Z 81.232,A 44.96824,B 0.00000,C 180.00000} ; preinsert
  LIN {X 15614.878,Y 985.187,Z -168.768,A 44.96824,B 0.00000,C 180.00000} ; insert
  LIN {X 15614.878,Y 985.187,Z -168.768,A 44.96824,B 0.00000,C 180.00000} ; release
  LIN {X 15614.878,Y 985.187,Z 131.232,A 44.96824,B 0.00000,C 180.00000} ; retreat
  ; Step 330, bar 3334
  LIN {X -15485.122,Y 985.187,Z 914.288,A 44.96824,B 0.00000,C 180.00000} ; outside
  LIN {X -15485.122,Y 985.187,Z 81.232,A 44.96824,B 0.00000,C 180.00000} ; preinsert
  LIN {X -15485.122,Y 985.187,Z -168.768,A 44.96824,B 0.00000,C 180.00000} ; insert
  LIN {X -15485.122,Y 985.187,Z -168.768,A 44.96824,B 0.00000,C 180.00000} ; release
  LIN {X -15485.122,Y 985.187,Z 131.232,A 44.96824,B 0.00000,C 180.00000} ; retreat
  ; Step 331, bar 3414
  LIN {X 15485.122,Y 985.187,Z 914.125,A 135.03176,B 0.00000,C 180.00000} ; outside
  LIN {X 15485.122,Y 985.187,Z 81.232,A 135.03176,B 0.00000,C 180.00000} ; preinsert
  LIN {X 15485.122,Y 985.187,Z -168.768,A 135.03176,B 0.00000,C 180.00000} ; insert
  LIN {X 15485.122,Y 985.187,Z -168.768,A 135.03176,B 0.00000,C 180.00000} ; release
  LIN {X 15485.122,Y 985.187,Z 131.232,A 135.03176,B 0.00000,C 180.00000} ; retreat
  ; Step 332, bar 3335
  LIN {X -15614.813,Y 1114.878,Z 914.125,A 45.03176,B 0.00000,C 180.00000} ; outside
  LIN {X -15614.813,Y 1114.878,Z 81.232,A 45.03176,B 0.00000,C 180.00000} ; preinsert
  LIN {X -15614.813,Y 1114.878,Z -168.768,A 45.03176,B 0.00000,C 180.00000} ; insert
  LIN {X -15614.813,Y 1114.878,Z -168.768,A 45.03176,B 0.00000,C 180.00000} ; release
  LIN {X -15614.813,Y 1114.878,Z 131.232,A 45.03176,B 0.00000,C 180.00000} ; retreat
  ; Step 333, bar 3415
  LIN {X 15614.813,Y 1114.878,Z 914.288,A 134.96824,B 0.00000,C 180.00000} ; outside
  LIN {X 15614.813,Y 1114.878,Z 81.232,A 134.96824,B 0.00000,C 180.00000} ; preinsert
  LIN {X 15614.813,Y 1114.878,Z -168.768,A 134.96824,B 0.00000,C 180.00000} ; insert
  LIN {X 15614.813,Y 1114.878,Z -168.768,A 134.96824,B 0.00000,C 180.00000} ; release
  LIN {X 15614.813,Y 1114.878,Z 131.232,A 134.96824,B 0.00000,C 180.00000} ; retreat
  ; Step 334, bar 3333
  LIN {X -15485.187,Y 1114.878,Z 914.288,A 134.96824,B 0.00000,C 180.00000} ; outside
  LIN {X -15485.187,Y 1114.878,Z 81.232,A 134.96824,B 0.00000,C 180.00000} ; preinsert
  LIN {X -15485.187,Y 1114.878,Z -168.768,A 134.96824,B 0.00000,C 180.00000} ; insert
  LIN {X -15485.187,Y 1114.878,Z -168.768,A 134.96824,B 0.00000,C 180.00000} ; release
  LIN {X -15485.187,Y 1114.878,Z 131.232,A 134.96824,B 0.00000,C 180.00000} ; retreat
  ; Step 335, bar 3413
  LIN {X 15485.187,Y 1114.878,Z 914.125,A 45.03176,B 0.00000,C 180.00000} ; outside
  LIN {X 15485.187,Y 1114.878,Z 81.232,A 45.03176,B 0.00000,C 180.00000} ; preinsert
  LIN {X 15485.187,Y 1114.878,Z -168.768,A 45.03176,B 0.00000,C 180.00000} ; insert
  LIN {X 15485.187,Y 1114.878,Z -168.768,A 45.03176,B 0.00000,C 180.00000} ; release
  LIN {X 15485.187,Y 1114.878,Z 131.232,A 45.03176,B 0.00000,C 180.00000} ; retreat
  ; Step 336, bar 3273
  LIN {X -14485.187,Y -1114.878,Z 914.125,A -134.96824,B 0.00000,C -180.00000} ; outside
  LIN {X -14485.187,Y -1114.878,Z 81.232,A -134.96824,B 0.00000,C -180.00000} ; preinsert
  LIN {X -14485.187,Y -1114.878,Z -168.768,A -134.96824,B 0.00000,C -180.00000} ; insert
  LIN {X -14485.187,Y -1114.878,Z -168.768,A -134.96824,B 0.00000,C -180.00000} ; release
  LIN {X -14485.187,Y -1114.878,Z 131.232,A -134.96824,B 0.00000,C -180.00000} ; retreat
  ; Step 337, bar 3275
  LIN {X -14614.813,Y -1114.878,Z 914.288,A -45.03176,B 0.00000,C 180.00000} ; outside
  LIN {X -14614.813,Y -1114.878,Z 81.232,A -45.03176,B 0.00000,C 180.00000} ; preinsert
  LIN {X -14614.813,Y -1114.878,Z -168.768,A -45.03176,B 0.00000,C 180.00000} ; insert
  LIN {X -14614.813,Y -1114.878,Z -168.768,A -45.03176,B 0.00000,C 180.00000} ; release
  LIN {X -14614.813,Y -1114.878,Z 131.232,A -45.03176,B 0.00000,C 180.00000} ; retreat
  ; Step 338, bar 3353
  LIN {X 14485.187,Y -1114.878,Z 914.288,A -45.03176,B 0.00000,C 180.00000} ; outside
  LIN {X 14485.187,Y -1114.878,Z 81.232,A -45.03176,B 0.00000,C 180.00000} ; preinsert
  LIN {X 14485.187,Y -1114.878,Z -168.768,A -45.03176,B 0.00000,C 180.00000} ; insert
  LIN {X 14485.187,Y -1114.878,Z -168.768,A -45.03176,B 0.00000,C 180.00000} ; release
  LIN {X 14485.187,Y -1114.878,Z 131.232,A -45.03176,B 0.00000,C 180.00000} ; retreat
  ; Step 339, bar 3355
  LIN {X 14614.813,Y -1114.878,Z 914.125,A -134.96824,B 0.00000,C -180.00000} ; outside
  LIN {X 14614.813,Y -1114.878,Z 81.232,A -134.96824,B 0.00000,C -180.00000} ; preinsert
  LIN {X 14614.813,Y -1114.878,Z -168.768,A -134.96824,B 0.00000,C -180.00000} ; insert
  LIN {X 14614.813,Y -1114.878,Z -168.768,A -134.96824,B 0.00000,C -180.00000} ; release
  LIN {X 14614.813,Y -1114.878,Z 131.232,A -134.96824,B 0.00000,C -180.00000} ; retreat
  ; Step 340, bar 3274
  LIN {X -14485.122,Y -985.187,Z 914.125,A -44.96824,B 0.00000,C 180.00000} ; outside
  LIN {X -14485.122,Y -985.187,Z 81.232,A -44.96824,B 0.00000,C 180.00000} ; preinsert
  LIN {X -14485.122,Y -985.187,Z -168.768,A -44.96824,B 0.00000,C 180.00000} ; insert
  LIN {X -14485.122,Y -985.187,Z -168.768,A -44.96824,B 0.00000,C 180.00000} ; release
  LIN {X -14485.122,Y -985.187,Z 131.232,A -44.96824,B 0.00000,C 180.00000} ; retreat
  ; Step 341, bar 3272
  LIN {X -14614.878,Y -985.187,Z 914.288,A -135.03176,B 0.00000,C -180.00000} ; outside
  LIN {X -14614.878,Y -985.187,Z 81.232,A -135.03176,B 0.00000,C -180.00000} ; preinsert
  LIN {X -14614.878,Y -985.187,Z -168.768,A -135.03176,B 0.00000,C -180.00000} ; insert
  LIN {X -14614.878,Y -985.187,Z -168.768,A -135.03176,B 0.00000,C -180.00000} ; release
  LIN {X -14614.878,Y -985.187,Z 131.232,A -135.03176,B 0.00000,C -180.00000} ; retreat
  ; Step 342, bar 3354
  LIN {X 14485.122,Y -985.187,Z 914.288,A -135.03176,B 0.00000,C 180.00000} ; outside
  LIN {X 14485.122,Y -985.187,Z 81.232,A -135.03176,B 0.00000,C 180.00000} ; preinsert
  LIN {X 14485.122,Y -985.187,Z -168.768,A -135.03176,B 0.00000,C 180.00000} ; insert
  LIN {X 14485.122,Y -985.187,Z -168.768,A -135.03176,B 0.00000,C 180.00000} ; release
  LIN {X 14485.122,Y -985.187,Z 131.232,A -135.03176,B 0.00000,C 180.00000} ; retreat
  ; Step 343, bar 3352
  LIN {X 14614.878,Y -985.187,Z 914.125,A -44.96824,B 0.00000,C 180.00000} ; outside
  LIN {X 14614.878,Y -985.187,Z 81.232,A -44.96824,B 0.00000,C 180.00000} ; preinsert
  LIN {X 14614.878,Y -985.187,Z -168.768,A -44.96824,B 0.00000,C 180.00000} ; insert
  LIN {X 14614.878,Y -985.187,Z -168.768,A -44.96824,B 0.00000,C 180.00000} ; release
  LIN {X 14614.878,Y -985.187,Z 131.232,A -44.96824,B 0.00000,C 180.00000} ; retreat
  ; Step 344, bar 3312
  LIN {X -14614.878,Y 985.187,Z 914.125,A 135.03176,B 0.00000,C 180.00000} ; outside
  LIN {X -14614.878,Y 985.187,Z 81.232,A 135.03176,B 0.00000,C 180.00000} ; preinsert
  LIN {X -14614.878,Y 985.187,Z -168.768,A 135.03176,B 0.00000,C 180.00000} ; insert
  LIN {X -14614.878,Y 985.187,Z -168.768,A 135.03176,B 0.00000,C 180.00000} ; release
  LIN {X -14614.878,Y 985.187,Z 131.232,A 135.03176,B 0.00000,C 180.00000} ; retreat
  ; Step 345, bar 3392
  LIN {X 14614.878,Y 985.187,Z 914.288,A 44.96824,B 0.00000,C 180.00000} ; outside
  LIN {X 14614.878,Y 985.187,Z 81.232,A 44.96824,B 0.00000,C 180.00000} ; preinsert
  LIN {X 14614.878,Y 985.187,Z -168.768,A 44.96824,B 0.00000,C 180.00000} ; insert
  LIN {X 14614.878,Y 985.187,Z -168.768,A 44.96824,B 0.00000,C 180.00000} ; release
  LIN {X 14614.878,Y 985.187,Z 131.232,A 44.96824,B 0.00000,C 180.00000} ; retreat
  ; Step 346, bar 3314
  LIN {X -14485.122,Y 985.187,Z 914.288,A 44.96824,B 0.00000,C 180.00000} ; outside
  LIN {X -14485.122,Y 985.187,Z 81.232,A 44.96824,B 0.00000,C 180.00000} ; preinsert
  LIN {X -14485.122,Y 985.187,Z -168.768,A 44.96824,B 0.00000,C 180.00000} ; insert
  LIN {X -14485.122,Y 985.187,Z -168.768,A 44.96824,B 0.00000,C 180.00000} ; release
  LIN {X -14485.122,Y 985.187,Z 131.232,A 44.96824,B 0.00000,C 180.00000} ; retreat
  ; Step 347, bar 3394
  LIN {X 14485.122,Y 985.187,Z 914.125,A 135.03176,B 0.00000,C 180.00000} ; outside
  LIN {X 14485.122,Y 985.187,Z 81.232,A 135.03176,B 0.00000,C 180.00000} ; preinsert
  LIN {X 14485.122,Y 985.187,Z -168.768,A 135.03176,B 0.00000,C 180.00000} ; insert
  LIN {X 14485.122,Y 985.187,Z -168.768,A 135.03176,B 0.00000,C 180.00000} ; release
  LIN {X 14485.122,Y 985.187,Z 131.232,A 135.03176,B 0.00000,C 180.00000} ; retreat
  ; Step 348, bar 3315
  LIN {X -14614.813,Y 1114.878,Z 914.125,A 45.03176,B 0.00000,C 180.00000} ; outside
  LIN {X -14614.813,Y 1114.878,Z 81.232,A 45.03176,B 0.00000,C 180.00000} ; preinsert
  LIN {X -14614.813,Y 1114.878,Z -168.768,A 45.03176,B 0.00000,C 180.00000} ; insert
  LIN {X -14614.813,Y 1114.878,Z -168.768,A 45.03176,B 0.00000,C 180.00000} ; release
  LIN {X -14614.813,Y 1114.878,Z 131.232,A 45.03176,B 0.00000,C 180.00000} ; retreat
  ; Step 349, bar 3395
  LIN {X 14614.813,Y 1114.878,Z 914.288,A 134.96824,B 0.00000,C 180.00000} ; outside
  LIN {X 14614.813,Y 1114.878,Z 81.232,A 134.96824,B 0.00000,C 180.00000} ; preinsert
  LIN {X 14614.813,Y 1114.878,Z -168.768,A 134.96824,B 0.00000,C 180.00000} ; insert
  LIN {X 14614.813,Y 1114.878,Z -168.768,A 134.96824,B 0.00000,C 180.00000} ; release
  LIN {X 14614.813,Y 1114.878,Z 131.232,A 134.96824,B 0.00000,C 180.00000} ; retreat
  ; Step 350, bar 3313
  LIN {X -14485.187,Y 1114.878,Z 914.288,A 134.96824,B 0.00000,C 180.00000} ; outside
  LIN {X -14485.187,Y 1114.878,Z 81.232,A 134.96824,B 0.00000,C 180.00000} ; preinsert
  LIN {X -14485.187,Y 1114.878,Z -168.768,A 134.96824,B 0.00000,C 180.00000} ; insert
  LIN {X -14485.187,Y 1114.878,Z -168.768,A 134.96824,B 0.00000,C 180.00000} ; release
  LIN {X -14485.187,Y 1114.878,Z 131.232,A 134.96824,B 0.00000,C 180.00000} ; retreat
  ; Step 351, bar 3393
  LIN {X 14485.187,Y 1114.878,Z 914.125,A 45.03176,B 0.00000,C 180.00000} ; outside
  LIN {X 14485.187,Y 1114.878,Z 81.232,A 45.03176,B 0.00000,C 180.00000} ; preinsert
  LIN {X 14485.187,Y 1114.878,Z -168.768,A 45.03176,B 0.00000,C 180.00000} ; insert
  LIN {X 14485.187,Y 1114.878,Z -168.768,A 45.03176,B 0.00000,C 180.00000} ; release
  LIN {X 14485.187,Y 1114.878,Z 131.232,A 45.03176,B 0.00000,C 180.00000} ; retreat
  ; Step 352, bar 1243
  LIN {X -13349.921,Y 0.110,Z 792.800,A 89.99666,B 0.00000,C 180.00000} ; outside
  LIN {X -13349.921,Y 0.110,Z -43.033,A 89.99666,B 0.00000,C 180.00000} ; preinsert
  LIN {X -13349.921,Y 0.110,Z -293.033,A 89.99666,B 0.00000,C 180.00000} ; insert
  LIN {X -13349.921,Y 0.110,Z -293.033,A 89.99666,B 0.00000,C 180.00000} ; release
  LIN {X -13349.921,Y 0.110,Z 6.967,A 89.99666,B 0.00000,C 180.00000} ; retreat
  ; Step 353, bar 1028
  LIN {X 13349.921,Y 0.097,Z 792.800,A 90.00334,B 0.00000,C 180.00000} ; outside
  LIN {X 13349.921,Y 0.097,Z -43.033,A 90.00334,B 0.00000,C 180.00000} ; preinsert
  LIN {X 13349.921,Y 0.097,Z -293.033,A 90.00334,B 0.00000,C 180.00000} ; insert
  LIN {X 13349.921,Y 0.097,Z -293.033,A 90.00334,B 0.00000,C 180.00000} ; release
  LIN {X 13349.921,Y 0.097,Z 6.967,A 90.00334,B 0.00000,C 180.00000} ; retreat
  ; Step 354, bar 1249
  LIN {X -13265.921,Y 0.110,Z 805.775,A 89.99666,B 0.00000,C 180.00000} ; outside
  LIN {X -13265.921,Y 0.110,Z -36.352,A 89.99666,B 0.00000,C 180.00000} ; preinsert
  LIN {X -13265.921,Y 0.110,Z -286.352,A 89.99666,B 0.00000,C 180.00000} ; insert
  LIN {X -13265.921,Y 0.110,Z -286.352,A 89.99666,B 0.00000,C 180.00000} ; release
  LIN {X -13265.921,Y 0.110,Z 13.648,A 89.99666,B 0.00000,C 180.00000} ; retreat
  ; Step 355, bar 1242
  LIN {X -13249.921,Y 0.110,Z 805.775,A 89.99666,B 0.00000,C 180.00000} ; outside
  LIN {X -13249.921,Y 0.110,Z -36.352,A 89.99666,B 0.00000,C 180.00000} ; preinsert
  LIN {X -13249.921,Y 0.110,Z -286.352,A 89.99666,B 0.00000,C 180.00000} ; insert
  LIN {X -13249.921,Y 0.110,Z -286.352,A 89.99666,B 0.00000,C 180.00000} ; release
  LIN {X -13249.921,Y 0.110,Z 13.648,A 89.99666,B 0.00000,C 180.00000} ; retreat
  ; Step 356, bar 1027
  LIN {X 13249.921,Y 0.097,Z 805.775,A 90.00334,B 0.00000,C 180.00000} ; outside
  LIN {X 13249.921,Y 0.097,Z -36.352,A 90.00334,B 0.00000,C 180.00000} ; preinsert
  LIN {X 13249.921,Y 0.097,Z -286.352,A 90.00334,B 0.00000,C 180.00000} ; insert
  LIN {X 13249.921,Y 0.097,Z -286.352,A 90.00334,B 0.00000,C 180.00000} ; release
  LIN {X 13249.921,Y 0.097,Z 13.648,A 90.00334,B 0.00000,C 180.00000} ; retreat
  ; Step 357, bar 1035
  LIN {X 13265.921,Y 0.097,Z 805.775,A 90.00334,B 0.00000,C 180.00000} ; outside
  LIN {X 13265.921,Y 0.097,Z -36.352,A 90.00334,B 0.00000,C 180.00000} ; preinsert
  LIN {X 13265.921,Y 0.097,Z -286.352,A 90.00334,B 0.00000,C 180.00000} ; insert
  LIN {X 13265.921,Y 0.097,Z -286.352,A 90.00334,B 0.00000,C 180.00000} ; release
  LIN {X 13265.921,Y 0.097,Z 13.648,A 90.00334,B 0.00000,C 180.00000} ; retreat
  ; Step 358, bar 3196
  LIN {X -14073.123,Y -2173.194,Z 947.594,A 134.95763,B 0.00000,C 180.00000} ; outside
  LIN {X -14073.123,Y -2173.194,Z 98.038,A 134.95763,B 0.00000,C 180.00000} ; preinsert
  LIN {X -14073.123,Y -2173.194,Z -151.962,A 134.95763,B 0.00000,C 180.00000} ; insert
  LIN {X -14073.123,Y -2173.194,Z -151.962,A 134.95763,B 0.00000,C 180.00000} ; release
  LIN {X -14073.123,Y -2173.194,Z 148.038,A 134.95763,B 0.00000,C 180.00000} ; retreat
  ; Step 359, bar 3198
  LIN {X -13926.877,Y -2173.194,Z 947.644,A 45.04237,B 0.00000,C 180.00000} ; outside
  LIN {X -13926.877,Y -2173.194,Z 98.038,A 45.04237,B 0.00000,C 180.00000} ; preinsert
  LIN {X -13926.877,Y -2173.194,Z -151.962,A 45.04237,B 0.00000,C 180.00000} ; insert
  LIN {X -13926.877,Y -2173.194,Z -151.962,A 45.04237,B 0.00000,C 180.00000} ; release
  LIN {X -13926.877,Y -2173.194,Z 148.038,A 45.04237,B 0.00000,C 180.00000} ; retreat
  ; Step 360, bar 3204
  LIN {X -10073.123,Y -2173.194,Z 947.594,A 134.95763,B 0.00000,C 180.00000} ; outside
  LIN {X -10073.123,Y -2173.194,Z 98.038,A 134.95763,B 0.00000,C 180.00000} ; preinsert
  LIN {X -10073.123,Y -2173.194,Z -151.962,A 134.95763,B 0.00000,C 180.00000} ; insert
  LIN {X -10073.123,Y -2173.194,Z -151.962,A 134.95763,B 0.00000,C 180.00000} ; release
  LIN {X -10073.123,Y -2173.194,Z 148.038,A 134.95763,B 0.00000,C 180.00000} ; retreat
  ; Step 361, bar 3206
  LIN {X -9926.877,Y -2173.194,Z 947.644,A 45.04237,B 0.00000,C 180.00000} ; outside
  LIN {X -9926.877,Y -2173.194,Z 98.038,A 45.04237,B 0.00000,C 180.00000} ; preinsert
  LIN {X -9926.877,Y -2173.194,Z -151.962,A 45.04237,B 0.00000,C 180.00000} ; insert
  LIN {X -9926.877,Y -2173.194,Z -151.962,A 45.04237,B 0.00000,C 180.00000} ; release
  LIN {X -9926.877,Y -2173.194,Z 148.038,A 45.04237,B 0.00000,C 180.00000} ; retreat
  ; Step 362, bar 3212
  LIN {X -6073.123,Y -2173.194,Z 947.594,A 134.95763,B 0.00000,C 180.00000} ; outside
  LIN {X -6073.123,Y -2173.194,Z 98.038,A 134.95763,B 0.00000,C 180.00000} ; preinsert
  LIN {X -6073.123,Y -2173.194,Z -151.962,A 134.95763,B 0.00000,C 180.00000} ; insert
  LIN {X -6073.123,Y -2173.194,Z -151.962,A 134.95763,B 0.00000,C 180.00000} ; release
  LIN {X -6073.123,Y -2173.194,Z 148.038,A 134.95763,B 0.00000,C 180.00000} ; retreat
  ; Step 363, bar 3214
  LIN {X -5926.877,Y -2173.194,Z 947.644,A 45.04237,B 0.00000,C 180.00000} ; outside
  LIN {X -5926.877,Y -2173.194,Z 98.038,A 45.04237,B 0.00000,C 180.00000} ; preinsert
  LIN {X -5926.877,Y -2173.194,Z -151.962,A 45.04237,B 0.00000,C 180.00000} ; insert
  LIN {X -5926.877,Y -2173.194,Z -151.962,A 45.04237,B 0.00000,C 180.00000} ; release
  LIN {X -5926.877,Y -2173.194,Z 148.038,A 45.04237,B 0.00000,C 180.00000} ; retreat
  ; Step 364, bar 3220
  LIN {X -2073.121,Y -2173.194,Z 947.594,A 134.95763,B 0.00000,C -180.00000} ; outside
  LIN {X -2073.121,Y -2173.194,Z 98.038,A 134.95763,B 0.00000,C -180.00000} ; preinsert
  LIN {X -2073.121,Y -2173.194,Z -151.962,A 134.95763,B 0.00000,C -180.00000} ; insert
  LIN {X -2073.121,Y -2173.194,Z -151.962,A 134.95763,B 0.00000,C -180.00000} ; release
  LIN {X -2073.121,Y -2173.194,Z 148.038,A 134.95763,B 0.00000,C -180.00000} ; retreat
  ; Step 365, bar 3222
  LIN {X -1926.875,Y -2173.194,Z 947.644,A 45.04237,B 0.00000,C 180.00000} ; outside
  LIN {X -1926.875,Y -2173.194,Z 98.038,A 45.04237,B 0.00000,C 180.00000} ; preinsert
  LIN {X -1926.875,Y -2173.194,Z -151.962,A 45.04237,B 0.00000,C 180.00000} ; insert
  LIN {X -1926.875,Y -2173.194,Z -151.962,A 45.04237,B 0.00000,C 180.00000} ; release
  LIN {X -1926.875,Y -2173.194,Z 148.038,A 45.04237,B 0.00000,C 180.00000} ; retreat
  ; Step 366, bar 3228
  LIN {X 1926.879,Y -2173.194,Z 947.594,A 134.95763,B 0.00000,C -180.00000} ; outside
  LIN {X 1926.879,Y -2173.194,Z 98.038,A 134.95763,B 0.00000,C -180.00000} ; preinsert
  LIN {X 1926.879,Y -2173.194,Z -151.962,A 134.95763,B 0.00000,C -180.00000} ; insert
  LIN {X 1926.879,Y -2173.194,Z -151.962,A 134.95763,B 0.00000,C -180.00000} ; release
  LIN {X 1926.879,Y -2173.194,Z 148.038,A 134.95763,B 0.00000,C -180.00000} ; retreat
  ; Step 367, bar 3230
  LIN {X 2073.125,Y -2173.194,Z 947.644,A 45.04237,B 0.00000,C 180.00000} ; outside
  LIN {X 2073.125,Y -2173.194,Z 98.038,A 45.04237,B 0.00000,C 180.00000} ; preinsert
  LIN {X 2073.125,Y -2173.194,Z -151.962,A 45.04237,B 0.00000,C 180.00000} ; insert
  LIN {X 2073.125,Y -2173.194,Z -151.962,A 45.04237,B 0.00000,C 180.00000} ; release
  LIN {X 2073.125,Y -2173.194,Z 148.038,A 45.04237,B 0.00000,C 180.00000} ; retreat
  ; Step 368, bar 3236
  LIN {X 5926.879,Y -2173.194,Z 947.594,A 134.95763,B 0.00000,C 180.00000} ; outside
  LIN {X 5926.879,Y -2173.194,Z 98.038,A 134.95763,B 0.00000,C 180.00000} ; preinsert
  LIN {X 5926.879,Y -2173.194,Z -151.962,A 134.95763,B 0.00000,C 180.00000} ; insert
  LIN {X 5926.879,Y -2173.194,Z -151.962,A 134.95763,B 0.00000,C 180.00000} ; release
  LIN {X 5926.879,Y -2173.194,Z 148.038,A 134.95763,B 0.00000,C 180.00000} ; retreat
  ; Step 369, bar 3238
  LIN {X 6073.125,Y -2173.194,Z 947.644,A 45.04237,B 0.00000,C 180.00000} ; outside
  LIN {X 6073.125,Y -2173.194,Z 98.038,A 45.04237,B 0.00000,C 180.00000} ; preinsert
  LIN {X 6073.125,Y -2173.194,Z -151.962,A 45.04237,B 0.00000,C 180.00000} ; insert
  LIN {X 6073.125,Y -2173.194,Z -151.962,A 45.04237,B 0.00000,C 180.00000} ; release
  LIN {X 6073.125,Y -2173.194,Z 148.038,A 45.04237,B 0.00000,C 180.00000} ; retreat
  ; Step 370, bar 3244
  LIN {X 9926.879,Y -2173.194,Z 947.594,A 134.95763,B 0.00000,C 180.00000} ; outside
  LIN {X 9926.879,Y -2173.194,Z 98.038,A 134.95763,B 0.00000,C 180.00000} ; preinsert
  LIN {X 9926.879,Y -2173.194,Z -151.962,A 134.95763,B 0.00000,C 180.00000} ; insert
  LIN {X 9926.879,Y -2173.194,Z -151.962,A 134.95763,B 0.00000,C 180.00000} ; release
  LIN {X 9926.879,Y -2173.194,Z 148.038,A 134.95763,B 0.00000,C 180.00000} ; retreat
  ; Step 371, bar 3246
  LIN {X 10073.125,Y -2173.194,Z 947.644,A 45.04237,B 0.00000,C 180.00000} ; outside
  LIN {X 10073.125,Y -2173.194,Z 98.038,A 45.04237,B 0.00000,C 180.00000} ; preinsert
  LIN {X 10073.125,Y -2173.194,Z -151.962,A 45.04237,B 0.00000,C 180.00000} ; insert
  LIN {X 10073.125,Y -2173.194,Z -151.962,A 45.04237,B 0.00000,C 180.00000} ; release
  LIN {X 10073.125,Y -2173.194,Z 148.038,A 45.04237,B 0.00000,C 180.00000} ; retreat
  ; Step 372, bar 3252
  LIN {X 13926.879,Y -2173.194,Z 947.594,A 134.95763,B 0.00000,C 180.00000} ; outside
  LIN {X 13926.879,Y -2173.194,Z 98.038,A 134.95763,B 0.00000,C 180.00000} ; preinsert
  LIN {X 13926.879,Y -2173.194,Z -151.962,A 134.95763,B 0.00000,C 180.00000} ; insert
  LIN {X 13926.879,Y -2173.194,Z -151.962,A 134.95763,B 0.00000,C 180.00000} ; release
  LIN {X 13926.879,Y -2173.194,Z 148.038,A 134.95763,B 0.00000,C 180.00000} ; retreat
  ; Step 373, bar 3254
  LIN {X 14073.125,Y -2173.194,Z 947.644,A 45.04237,B 0.00000,C 180.00000} ; outside
  LIN {X 14073.125,Y -2173.194,Z 98.038,A 45.04237,B 0.00000,C 180.00000} ; preinsert
  LIN {X 14073.125,Y -2173.194,Z -151.962,A 45.04237,B 0.00000,C 180.00000} ; insert
  LIN {X 14073.125,Y -2173.194,Z -151.962,A 45.04237,B 0.00000,C 180.00000} ; release
  LIN {X 14073.125,Y -2173.194,Z 148.038,A 45.04237,B 0.00000,C 180.00000} ; retreat
  ; Step 374, bar 3197
  LIN {X -14073.194,Y -2026.877,Z 947.594,A 44.95763,B 0.00000,C 180.00000} ; outside
  LIN {X -14073.194,Y -2026.877,Z 98.038,A 44.95763,B 0.00000,C 180.00000} ; preinsert
  LIN {X -14073.194,Y -2026.877,Z -151.962,A 44.95763,B 0.00000,C 180.00000} ; insert
  LIN {X -14073.194,Y -2026.877,Z -151.962,A 44.95763,B 0.00000,C 180.00000} ; release
  LIN {X -14073.194,Y -2026.877,Z 148.038,A 44.95763,B 0.00000,C 180.00000} ; retreat
  ; Step 375, bar 3205
  LIN {X -10073.194,Y -2026.877,Z 947.594,A 44.95763,B 0.00000,C 180.00000} ; outside
  LIN {X -10073.194,Y -2026.877,Z 98.038,A 44.95763,B 0.00000,C 180.00000} ; preinsert
  LIN {X -10073.194,Y -2026.877,Z -151.962,A 44.95763,B 0.00000,C 180.00000} ; insert
  LIN {X -10073.194,Y -2026.877,Z -151.962,A 44.95763,B 0.00000,C 180.00000} ; release
  LIN {X -10073.194,Y -2026.877,Z 148.038,A 44.95763,B 0.00000,C 180.00000} ; retreat
  ; Step 376, bar 3213
  LIN {X -6073.194,Y -2026.877,Z 947.594,A 44.95763,B 0.00000,C 180.00000} ; outside
  LIN {X -6073.194,Y -2026.877,Z 98.038,A 44.95763,B 0.00000,C 180.00000} ; preinsert
  LIN {X -6073.194,Y -2026.877,Z -151.962,A 44.95763,B 0.00000,C 180.00000} ; insert
  LIN {X -6073.194,Y -2026.877,Z -151.962,A 44.95763,B 0.00000,C 180.00000} ; release
  LIN {X -6073.194,Y -2026.877,Z 148.038,A 44.95763,B 0.00000,C 180.00000} ; retreat
  ; Step 377, bar 3221
  LIN {X -2073.193,Y -2026.877,Z 947.594,A 44.95763,B 0.00000,C 180.00000} ; outside
  LIN {X -2073.193,Y -2026.877,Z 98.038,A 44.95763,B 0.00000,C 180.00000} ; preinsert
  LIN {X -2073.193,Y -2026.877,Z -151.962,A 44.95763,B 0.00000,C 180.00000} ; insert
  LIN {X -2073.193,Y -2026.877,Z -151.962,A 44.95763,B 0.00000,C 180.00000} ; release
  LIN {X -2073.193,Y -2026.877,Z 148.038,A 44.95763,B 0.00000,C 180.00000} ; retreat
  ; Step 378, bar 3229
  LIN {X 1926.807,Y -2026.877,Z 947.594,A 44.95763,B 0.00000,C 180.00000} ; outside
  LIN {X 1926.807,Y -2026.877,Z 98.038,A 44.95763,B 0.00000,C 180.00000} ; preinsert
  LIN {X 1926.807,Y -2026.877,Z -151.962,A 44.95763,B 0.00000,C 180.00000} ; insert
  LIN {X 1926.807,Y -2026.877,Z -151.962,A 44.95763,B 0.00000,C 180.00000} ; release
  LIN {X 1926.807,Y -2026.877,Z 148.038,A 44.95763,B 0.00000,C 180.00000} ; retreat
  ; Step 379, bar 3237
  LIN {X 5926.807,Y -2026.877,Z 947.594,A 44.95763,B 0.00000,C 180.00000} ; outside
  LIN {X 5926.807,Y -2026.877,Z 98.038,A 44.95763,B 0.00000,C 180.00000} ; preinsert
  LIN {X 5926.807,Y -2026.877,Z -151.962,A 44.95763,B 0.00000,C 180.00000} ; insert
  LIN {X 5926.807,Y -2026.877,Z -151.962,A 44.95763,B 0.00000,C 180.00000} ; release
  LIN {X 5926.807,Y -2026.877,Z 148.038,A 44.95763,B 0.00000,C 180.00000} ; retreat
  ; Step 380, bar 3245
  LIN {X 9926.807,Y -2026.877,Z 947.594,A 44.95763,B 0.00000,C 180.00000} ; outside
  LIN {X 9926.807,Y -2026.877,Z 98.038,A 44.95763,B 0.00000,C 180.00000} ; preinsert
  LIN {X 9926.807,Y -2026.877,Z -151.962,A 44.95763,B 0.00000,C 180.00000} ; insert
  LIN {X 9926.807,Y -2026.877,Z -151.962,A 44.95763,B 0.00000,C 180.00000} ; release
  LIN {X 9926.807,Y -2026.877,Z 148.038,A 44.95763,B 0.00000,C 180.00000} ; retreat
  ; Step 381, bar 3253
  LIN {X 13926.807,Y -2026.877,Z 947.594,A 44.95763,B 0.00000,C 180.00000} ; outside
  LIN {X 13926.807,Y -2026.877,Z 98.038,A 44.95763,B 0.00000,C 180.00000} ; preinsert
  LIN {X 13926.807,Y -2026.877,Z -151.962,A 44.95763,B 0.00000,C 180.00000} ; insert
  LIN {X 13926.807,Y -2026.877,Z -151.962,A 44.95763,B 0.00000,C 180.00000} ; release
  LIN {X 13926.807,Y -2026.877,Z 148.038,A 44.95763,B 0.00000,C 180.00000} ; retreat
  ; Step 382, bar 3199
  LIN {X -13926.806,Y -2026.877,Z 947.644,A 135.04237,B 0.00000,C 180.00000} ; outside
  LIN {X -13926.806,Y -2026.877,Z 98.038,A 135.04237,B 0.00000,C 180.00000} ; preinsert
  LIN {X -13926.806,Y -2026.877,Z -151.962,A 135.04237,B 0.00000,C 180.00000} ; insert
  LIN {X -13926.806,Y -2026.877,Z -151.962,A 135.04237,B 0.00000,C 180.00000} ; release
  LIN {X -13926.806,Y -2026.877,Z 148.038,A 135.04237,B 0.00000,C 180.00000} ; retreat
  ; Step 383, bar 3207
  LIN {X -9926.806,Y -2026.877,Z 947.644,A 135.04237,B 0.00000,C 180.00000} ; outside
  LIN {X -9926.806,Y -2026.877,Z 98.038,A 135.04237,B 0.00000,C 180.00000} ; preinsert
  LIN {X -9926.806,Y -2026.877,Z -151.962,A 135.04237,B 0.00000,C 180.00000} ; insert
  LIN {X -9926.806,Y -2026.877,Z -151.962,A 135.04237,B 0.00000,C 180.00000} ; release
  LIN {X -9926.806,Y -2026.877,Z 148.038,A 135.04237,B 0.00000,C 180.00000} ; retreat
  ; Step 384, bar 3215
  LIN {X -5926.806,Y -2026.877,Z 947.644,A 135.04237,B 0.00000,C 180.00000} ; outside
  LIN {X -5926.806,Y -2026.877,Z 98.038,A 135.04237,B 0.00000,C 180.00000} ; preinsert
  LIN {X -5926.806,Y -2026.877,Z -151.962,A 135.04237,B 0.00000,C 180.00000} ; insert
  LIN {X -5926.806,Y -2026.877,Z -151.962,A 135.04237,B 0.00000,C 180.00000} ; release
  LIN {X -5926.806,Y -2026.877,Z 148.038,A 135.04237,B 0.00000,C 180.00000} ; retreat
  ; Step 385, bar 3223
  LIN {X -1926.804,Y -2026.877,Z 947.644,A 135.04237,B 0.00000,C 180.00000} ; outside
  LIN {X -1926.804,Y -2026.877,Z 98.038,A 135.04237,B 0.00000,C 180.00000} ; preinsert
  LIN {X -1926.804,Y -2026.877,Z -151.962,A 135.04237,B 0.00000,C 180.00000} ; insert
  LIN {X -1926.804,Y -2026.877,Z -151.962,A 135.04237,B 0.00000,C 180.00000} ; release
  LIN {X -1926.804,Y -2026.877,Z 148.038,A 135.04237,B 0.00000,C 180.00000} ; retreat
  ; Step 386, bar 3231
  LIN {X 2073.196,Y -2026.877,Z 947.644,A 135.04237,B 0.00000,C 180.00000} ; outside
  LIN {X 2073.196,Y -2026.877,Z 98.038,A 135.04237,B 0.00000,C 180.00000} ; preinsert
  LIN {X 2073.196,Y -2026.877,Z -151.962,A 135.04237,B 0.00000,C 180.00000} ; insert
  LIN {X 2073.196,Y -2026.877,Z -151.962,A 135.04237,B 0.00000,C 180.00000} ; release
  LIN {X 2073.196,Y -2026.877,Z 148.038,A 135.04237,B 0.00000,C 180.00000} ; retreat
  ; Step 387, bar 3239
  LIN {X 6073.196,Y -2026.877,Z 947.644,A 135.04237,B 0.00000,C 180.00000} ; outside
  LIN {X 6073.196,Y -2026.877,Z 98.038,A 135.04237,B 0.00000,C 180.00000} ; preinsert
  LIN {X 6073.196,Y -2026.877,Z -151.962,A 135.04237,B 0.00000,C 180.00000} ; insert
  LIN {X 6073.196,Y -2026.877,Z -151.962,A 135.04237,B 0.00000,C 180.00000} ; release
  LIN {X 6073.196,Y -2026.877,Z 148.038,A 135.04237,B 0.00000,C 180.00000} ; retreat
  ; Step 388, bar 3247
  LIN {X 10073.196,Y -2026.877,Z 947.644,A 135.04237,B 0.00000,C 180.00000} ; outside
  LIN {X 10073.196,Y -2026.877,Z 98.038,A 135.04237,B 0.00000,C 180.00000} ; preinsert
  LIN {X 10073.196,Y -2026.877,Z -151.962,A 135.04237,B 0.00000,C 180.00000} ; insert
  LIN {X 10073.196,Y -2026.877,Z -151.962,A 135.04237,B 0.00000,C 180.00000} ; release
  LIN {X 10073.196,Y -2026.877,Z 148.038,A 135.04237,B 0.00000,C 180.00000} ; retreat
  ; Step 389, bar 3255
  LIN {X 14073.196,Y -2026.877,Z 947.644,A 135.04237,B 0.00000,C 180.00000} ; outside
  LIN {X 14073.196,Y -2026.877,Z 98.038,A 135.04237,B 0.00000,C 180.00000} ; preinsert
  LIN {X 14073.196,Y -2026.877,Z -151.962,A 135.04237,B 0.00000,C 180.00000} ; insert
  LIN {X 14073.196,Y -2026.877,Z -151.962,A 135.04237,B 0.00000,C 180.00000} ; release
  LIN {X 14073.196,Y -2026.877,Z 148.038,A 135.04237,B 0.00000,C 180.00000} ; retreat
  ; Step 390, bar 3191
  LIN {X 14073.196,Y 2026.877,Z 947.594,A -135.04237,B 0.00000,C 180.00000} ; outside
  LIN {X 14073.196,Y 2026.877,Z 98.038,A -135.04237,B 0.00000,C 180.00000} ; preinsert
  LIN {X 14073.196,Y 2026.877,Z -151.962,A -135.04237,B 0.00000,C 180.00000} ; insert
  LIN {X 14073.196,Y 2026.877,Z -151.962,A -135.04237,B 0.00000,C 180.00000} ; release
  LIN {X 14073.196,Y 2026.877,Z 148.038,A -135.04237,B 0.00000,C 180.00000} ; retreat
  ; Step 391, bar 3183
  LIN {X 10073.196,Y 2026.877,Z 947.594,A -135.04237,B 0.00000,C 180.00000} ; outside
  LIN {X 10073.196,Y 2026.877,Z 98.038,A -135.04237,B 0.00000,C 180.00000} ; preinsert
  LIN {X 10073.196,Y 2026.877,Z -151.962,A -135.04237,B 0.00000,C 180.00000} ; insert
  LIN {X 10073.196,Y 2026.877,Z -151.962,A -135.04237,B 0.00000,C 180.00000} ; release
  LIN {X 10073.196,Y 2026.877,Z 148.038,A -135.04237,B 0.00000,C 180.00000} ; retreat
  ; Step 392, bar 3175
  LIN {X 6073.196,Y 2026.877,Z 947.594,A -135.04237,B 0.00000,C -180.00000} ; outside
  LIN {X 6073.196,Y 2026.877,Z 98.038,A -135.04237,B 0.00000,C -180.00000} ; preinsert
  LIN {X 6073.196,Y 2026.877,Z -151.962,A -135.04237,B 0.00000,C -180.00000} ; insert
  LIN {X 6073.196,Y 2026.877,Z -151.962,A -135.04237,B 0.00000,C -180.00000} ; release
  LIN {X 6073.196,Y 2026.877,Z 148.038,A -135.04237,B 0.00000,C -180.00000} ; retreat
  ; Step 393, bar 3167
  LIN {X 2073.196,Y 2026.877,Z 947.594,A -135.04237,B 0.00000,C -180.00000} ; outside
  LIN {X 2073.196,Y 2026.877,Z 98.038,A -135.04237,B 0.00000,C -180.00000} ; preinsert
  LIN {X 2073.196,Y 2026.877,Z -151.962,A -135.04237,B 0.00000,C -180.00000} ; insert
  LIN {X 2073.196,Y 2026.877,Z -151.962,A -135.04237,B 0.00000,C -180.00000} ; release
  LIN {X 2073.196,Y 2026.877,Z 148.038,A -135.04237,B 0.00000,C -180.00000} ; retreat
  ; Step 394, bar 3159
  LIN {X -1926.804,Y 2026.877,Z 947.594,A -135.04237,B 0.00000,C -180.00000} ; outside
  LIN {X -1926.804,Y 2026.877,Z 98.038,A -135.04237,B 0.00000,C -180.00000} ; preinsert
  LIN {X -1926.804,Y 2026.877,Z -151.962,A -135.04237,B 0.00000,C -180.00000} ; insert
  LIN {X -1926.804,Y 2026.877,Z -151.962,A -135.04237,B 0.00000,C -180.00000} ; release
  LIN {X -1926.804,Y 2026.877,Z 148.038,A -135.04237,B 0.00000,C -180.00000} ; retreat
  ; Step 395, bar 3151
  LIN {X -5926.806,Y 2026.877,Z 947.594,A -135.04237,B 0.00000,C -180.00000} ; outside
  LIN {X -5926.806,Y 2026.877,Z 98.038,A -135.04237,B 0.00000,C -180.00000} ; preinsert
  LIN {X -5926.806,Y 2026.877,Z -151.962,A -135.04237,B 0.00000,C -180.00000} ; insert
  LIN {X -5926.806,Y 2026.877,Z -151.962,A -135.04237,B 0.00000,C -180.00000} ; release
  LIN {X -5926.806,Y 2026.877,Z 148.038,A -135.04237,B 0.00000,C -180.00000} ; retreat
  ; Step 396, bar 3143
  LIN {X -9926.806,Y 2026.877,Z 947.594,A -135.04237,B 0.00000,C -180.00000} ; outside
  LIN {X -9926.806,Y 2026.877,Z 98.038,A -135.04237,B 0.00000,C -180.00000} ; preinsert
  LIN {X -9926.806,Y 2026.877,Z -151.962,A -135.04237,B 0.00000,C -180.00000} ; insert
  LIN {X -9926.806,Y 2026.877,Z -151.962,A -135.04237,B 0.00000,C -180.00000} ; release
  LIN {X -9926.806,Y 2026.877,Z 148.038,A -135.04237,B 0.00000,C -180.00000} ; retreat
  ; Step 397, bar 3135
  LIN {X -13926.806,Y 2026.877,Z 947.594,A -135.04237,B 0.00000,C 180.00000} ; outside
  LIN {X -13926.806,Y 2026.877,Z 98.038,A -135.04237,B 0.00000,C 180.00000} ; preinsert
  LIN {X -13926.806,Y 2026.877,Z -151.962,A -135.04237,B 0.00000,C 180.00000} ; insert
  LIN {X -13926.806,Y 2026.877,Z -151.962,A -135.04237,B 0.00000,C 180.00000} ; release
  LIN {X -13926.806,Y 2026.877,Z 148.038,A -135.04237,B 0.00000,C 180.00000} ; retreat
  ; Step 398, bar 3189
  LIN {X 13926.808,Y 2026.877,Z 947.644,A -44.95763,B 0.00000,C 180.00000} ; outside
  LIN {X 13926.808,Y 2026.877,Z 98.038,A -44.95763,B 0.00000,C 180.00000} ; preinsert
  LIN {X 13926.808,Y 2026.877,Z -151.962,A -44.95763,B 0.00000,C 180.00000} ; insert
  LIN {X 13926.808,Y 2026.877,Z -151.962,A -44.95763,B 0.00000,C 180.00000} ; release
  LIN {X 13926.808,Y 2026.877,Z 148.038,A -44.95763,B 0.00000,C 180.00000} ; retreat
  ; Step 399, bar 3181
  LIN {X 9926.808,Y 2026.877,Z 947.644,A -44.95763,B 0.00000,C 180.00000} ; outside
  LIN {X 9926.808,Y 2026.877,Z 98.038,A -44.95763,B 0.00000,C 180.00000} ; preinsert
  LIN {X 9926.808,Y 2026.877,Z -151.962,A -44.95763,B 0.00000,C 180.00000} ; insert
  LIN {X 9926.808,Y 2026.877,Z -151.962,A -44.95763,B 0.00000,C 180.00000} ; release
  LIN {X 9926.808,Y 2026.877,Z 148.038,A -44.95763,B 0.00000,C 180.00000} ; retreat
  ; Step 400, bar 3173
  LIN {X 5926.808,Y 2026.877,Z 947.644,A -44.95763,B 0.00000,C 180.00000} ; outside
  LIN {X 5926.808,Y 2026.877,Z 98.038,A -44.95763,B 0.00000,C 180.00000} ; preinsert
  LIN {X 5926.808,Y 2026.877,Z -151.962,A -44.95763,B 0.00000,C 180.00000} ; insert
  LIN {X 5926.808,Y 2026.877,Z -151.962,A -44.95763,B 0.00000,C 180.00000} ; release
  LIN {X 5926.808,Y 2026.877,Z 148.038,A -44.95763,B 0.00000,C 180.00000} ; retreat
  ; Step 401, bar 3165
  LIN {X 1926.808,Y 2026.877,Z 947.644,A -44.95763,B 0.00000,C 180.00000} ; outside
  LIN {X 1926.808,Y 2026.877,Z 98.038,A -44.95763,B 0.00000,C 180.00000} ; preinsert
  LIN {X 1926.808,Y 2026.877,Z -151.962,A -44.95763,B 0.00000,C 180.00000} ; insert
  LIN {X 1926.808,Y 2026.877,Z -151.962,A -44.95763,B 0.00000,C 180.00000} ; release
  LIN {X 1926.808,Y 2026.877,Z 148.038,A -44.95763,B 0.00000,C 180.00000} ; retreat
  ; Step 402, bar 3157
  LIN {X -2073.192,Y 2026.877,Z 947.644,A -44.95763,B 0.00000,C 180.00000} ; outside
  LIN {X -2073.192,Y 2026.877,Z 98.038,A -44.95763,B 0.00000,C 180.00000} ; preinsert
  LIN {X -2073.192,Y 2026.877,Z -151.962,A -44.95763,B 0.00000,C 180.00000} ; insert
  LIN {X -2073.192,Y 2026.877,Z -151.962,A -44.95763,B 0.00000,C 180.00000} ; release
  LIN {X -2073.192,Y 2026.877,Z 148.038,A -44.95763,B 0.00000,C 180.00000} ; retreat
  ; Step 403, bar 3149
  LIN {X -6073.194,Y 2026.877,Z 947.644,A -44.95763,B 0.00000,C 180.00000} ; outside
  LIN {X -6073.194,Y 2026.877,Z 98.038,A -44.95763,B 0.00000,C 180.00000} ; preinsert
  LIN {X -6073.194,Y 2026.877,Z -151.962,A -44.95763,B 0.00000,C 180.00000} ; insert
  LIN {X -6073.194,Y 2026.877,Z -151.962,A -44.95763,B 0.00000,C 180.00000} ; release
  LIN {X -6073.194,Y 2026.877,Z 148.038,A -44.95763,B 0.00000,C 180.00000} ; retreat
  ; Step 404, bar 3141
  LIN {X -10073.194,Y 2026.877,Z 947.644,A -44.95763,B 0.00000,C 180.00000} ; outside
  LIN {X -10073.194,Y 2026.877,Z 98.038,A -44.95763,B 0.00000,C 180.00000} ; preinsert
  LIN {X -10073.194,Y 2026.877,Z -151.962,A -44.95763,B 0.00000,C 180.00000} ; insert
  LIN {X -10073.194,Y 2026.877,Z -151.962,A -44.95763,B 0.00000,C 180.00000} ; release
  LIN {X -10073.194,Y 2026.877,Z 148.038,A -44.95763,B 0.00000,C 180.00000} ; retreat
  ; Step 405, bar 3133
  LIN {X -14073.194,Y 2026.877,Z 947.644,A -44.95763,B 0.00000,C 180.00000} ; outside
  LIN {X -14073.194,Y 2026.877,Z 98.038,A -44.95763,B 0.00000,C 180.00000} ; preinsert
  LIN {X -14073.194,Y 2026.877,Z -151.962,A -44.95763,B 0.00000,C 180.00000} ; insert
  LIN {X -14073.194,Y 2026.877,Z -151.962,A -44.95763,B 0.00000,C 180.00000} ; release
  LIN {X -14073.194,Y 2026.877,Z 148.038,A -44.95763,B 0.00000,C 180.00000} ; retreat
  ; Step 406, bar 3190
  LIN {X 14073.125,Y 2173.194,Z 947.594,A -45.04237,B 0.00000,C 180.00000} ; outside
  LIN {X 14073.125,Y 2173.194,Z 98.038,A -45.04237,B 0.00000,C 180.00000} ; preinsert
  LIN {X 14073.125,Y 2173.194,Z -151.962,A -45.04237,B 0.00000,C 180.00000} ; insert
  LIN {X 14073.125,Y 2173.194,Z -151.962,A -45.04237,B 0.00000,C 180.00000} ; release
  LIN {X 14073.125,Y 2173.194,Z 148.038,A -45.04237,B 0.00000,C 180.00000} ; retreat
  ; Step 407, bar 3188
  LIN {X 13926.879,Y 2173.194,Z 947.644,A -134.95763,B 0.00000,C -180.00000} ; outside
  LIN {X 13926.879,Y 2173.194,Z 98.038,A -134.95763,B 0.00000,C -180.00000} ; preinsert
  LIN {X 13926.879,Y 2173.194,Z -151.962,A -134.95763,B 0.00000,C -180.00000} ; insert
  LIN {X 13926.879,Y 2173.194,Z -151.962,A -134.95763,B 0.00000,C -180.00000} ; release
  LIN {X 13926.879,Y 2173.194,Z 148.038,A -134.95763,B 0.00000,C -180.00000} ; retreat
  ; Step 408, bar 3182
  LIN {X 10073.125,Y 2173.194,Z 947.594,A -45.04237,B 0.00000,C 180.00000} ; outside
  LIN {X 10073.125,Y 2173.194,Z 98.038,A -45.04237,B 0.00000,C 180.00000} ; preinsert
  LIN {X 10073.125,Y 2173.194,Z -151.962,A -45.04237,B 0.00000,C 180.00000} ; insert
  LIN {X 10073.125,Y 2173.194,Z -151.962,A -45.04237,B 0.00000,C 180.00000} ; release
  LIN {X 10073.125,Y 2173.194,Z 148.038,A -45.04237,B 0.00000,C 180.00000} ; retreat
  ; Step 409, bar 3180
  LIN {X 9926.879,Y 2173.194,Z 947.644,A -134.95763,B 0.00000,C -180.00000} ; outside
  LIN {X 9926.879,Y 2173.194,Z 98.038,A -134.95763,B 0.00000,C -180.00000} ; preinsert
  LIN {X 9926.879,Y 2173.194,Z -151.962,A -134.95763,B 0.00000,C -180.00000} ; insert
  LIN {X 9926.879,Y 2173.194,Z -151.962,A -134.95763,B 0.00000,C -180.00000} ; release
  LIN {X 9926.879,Y 2173.194,Z 148.038,A -134.95763,B 0.00000,C -180.00000} ; retreat
  ; Step 410, bar 3174
  LIN {X 6073.125,Y 2173.194,Z 947.594,A -45.04237,B 0.00000,C 180.00000} ; outside
  LIN {X 6073.125,Y 2173.194,Z 98.038,A -45.04237,B 0.00000,C 180.00000} ; preinsert
  LIN {X 6073.125,Y 2173.194,Z -151.962,A -45.04237,B 0.00000,C 180.00000} ; insert
  LIN {X 6073.125,Y 2173.194,Z -151.962,A -45.04237,B 0.00000,C 180.00000} ; release
  LIN {X 6073.125,Y 2173.194,Z 148.038,A -45.04237,B 0.00000,C 180.00000} ; retreat
  ; Step 411, bar 3172
  LIN {X 5926.879,Y 2173.194,Z 947.644,A -134.95763,B 0.00000,C -180.00000} ; outside
  LIN {X 5926.879,Y 2173.194,Z 98.038,A -134.95763,B 0.00000,C -180.00000} ; preinsert
  LIN {X 5926.879,Y 2173.194,Z -151.962,A -134.95763,B 0.00000,C -180.00000} ; insert
  LIN {X 5926.879,Y 2173.194,Z -151.962,A -134.95763,B 0.00000,C -180.00000} ; release
  LIN {X 5926.879,Y 2173.194,Z 148.038,A -134.95763,B 0.00000,C -180.00000} ; retreat
  ; Step 412, bar 3166
  LIN {X 2073.125,Y 2173.194,Z 947.594,A -45.04237,B 0.00000,C 180.00000} ; outside
  LIN {X 2073.125,Y 2173.194,Z 98.038,A -45.04237,B 0.00000,C 180.00000} ; preinsert
  LIN {X 2073.125,Y 2173.194,Z -151.962,A -45.04237,B 0.00000,C 180.00000} ; insert
  LIN {X 2073.125,Y 2173.194,Z -151.962,A -45.04237,B 0.00000,C 180.00000} ; release
  LIN {X 2073.125,Y 2173.194,Z 148.038,A -45.04237,B 0.00000,C 180.00000} ; retreat
  ; Step 413, bar 3164
  LIN {X 1926.879,Y 2173.194,Z 947.644,A -134.95763,B 0.00000,C -180.00000} ; outside
  LIN {X 1926.879,Y 2173.194,Z 98.038,A -134.95763,B 0.00000,C -180.00000} ; preinsert
  LIN {X 1926.879,Y 2173.194,Z -151.962,A -134.95763,B 0.00000,C -180.00000} ; insert
  LIN {X 1926.879,Y 2173.194,Z -151.962,A -134.95763,B 0.00000,C -180.00000} ; release
  LIN {X 1926.879,Y 2173.194,Z 148.038,A -134.95763,B 0.00000,C -180.00000} ; retreat
  ; Step 414, bar 3158
  LIN {X -1926.875,Y 2173.194,Z 947.594,A -45.04237,B 0.00000,C 180.00000} ; outside
  LIN {X -1926.875,Y 2173.194,Z 98.038,A -45.04237,B 0.00000,C 180.00000} ; preinsert
  LIN {X -1926.875,Y 2173.194,Z -151.962,A -45.04237,B 0.00000,C 180.00000} ; insert
  LIN {X -1926.875,Y 2173.194,Z -151.962,A -45.04237,B 0.00000,C 180.00000} ; release
  LIN {X -1926.875,Y 2173.194,Z 148.038,A -45.04237,B 0.00000,C 180.00000} ; retreat
  ; Step 415, bar 3156
  LIN {X -2073.121,Y 2173.194,Z 947.644,A -134.95763,B 0.00000,C -180.00000} ; outside
  LIN {X -2073.121,Y 2173.194,Z 98.038,A -134.95763,B 0.00000,C -180.00000} ; preinsert
  LIN {X -2073.121,Y 2173.194,Z -151.962,A -134.95763,B 0.00000,C -180.00000} ; insert
  LIN {X -2073.121,Y 2173.194,Z -151.962,A -134.95763,B 0.00000,C -180.00000} ; release
  LIN {X -2073.121,Y 2173.194,Z 148.038,A -134.95763,B 0.00000,C -180.00000} ; retreat
  ; Step 416, bar 3150
  LIN {X -5926.877,Y 2173.194,Z 947.594,A -45.04237,B 0.00000,C 180.00000} ; outside
  LIN {X -5926.877,Y 2173.194,Z 98.038,A -45.04237,B 0.00000,C 180.00000} ; preinsert
  LIN {X -5926.877,Y 2173.194,Z -151.962,A -45.04237,B 0.00000,C 180.00000} ; insert
  LIN {X -5926.877,Y 2173.194,Z -151.962,A -45.04237,B 0.00000,C 180.00000} ; release
  LIN {X -5926.877,Y 2173.194,Z 148.038,A -45.04237,B 0.00000,C 180.00000} ; retreat
  ; Step 417, bar 3148
  LIN {X -6073.123,Y 2173.194,Z 947.644,A -134.95763,B 0.00000,C -180.00000} ; outside
  LIN {X -6073.123,Y 2173.194,Z 98.038,A -134.95763,B 0.00000,C -180.00000} ; preinsert
  LIN {X -6073.123,Y 2173.194,Z -151.962,A -134.95763,B 0.00000,C -180.00000} ; insert
  LIN {X -6073.123,Y 2173.194,Z -151.962,A -134.95763,B 0.00000,C -180.00000} ; release
  LIN {X -6073.123,Y 2173.194,Z 148.038,A -134.95763,B 0.00000,C -180.00000} ; retreat
  ; Step 418, bar 3142
  LIN {X -9926.877,Y 2173.194,Z 947.594,A -45.04237,B 0.00000,C 180.00000} ; outside
  LIN {X -9926.877,Y 2173.194,Z 98.038,A -45.04237,B 0.00000,C 180.00000} ; preinsert
  LIN {X -9926.877,Y 2173.194,Z -151.962,A -45.04237,B 0.00000,C 180.00000} ; insert
  LIN {X -9926.877,Y 2173.194,Z -151.962,A -45.04237,B 0.00000,C 180.00000} ; release
  LIN {X -9926.877,Y 2173.194,Z 148.038,A -45.04237,B 0.00000,C 180.00000} ; retreat
  ; Step 419, bar 3140
  LIN {X -10073.123,Y 2173.194,Z 947.644,A -134.95763,B 0.00000,C -180.00000} ; outside
  LIN {X -10073.123,Y 2173.194,Z 98.038,A -134.95763,B 0.00000,C -180.00000} ; preinsert
  LIN {X -10073.123,Y 2173.194,Z -151.962,A -134.95763,B 0.00000,C -180.00000} ; insert
  LIN {X -10073.123,Y 2173.194,Z -151.962,A -134.95763,B 0.00000,C -180.00000} ; release
  LIN {X -10073.123,Y 2173.194,Z 148.038,A -134.95763,B 0.00000,C -180.00000} ; retreat
  ; Step 420, bar 3134
  LIN {X -13926.877,Y 2173.194,Z 947.594,A -45.04237,B 0.00000,C 180.00000} ; outside
  LIN {X -13926.877,Y 2173.194,Z 98.038,A -45.04237,B 0.00000,C 180.00000} ; preinsert
  LIN {X -13926.877,Y 2173.194,Z -151.962,A -45.04237,B 0.00000,C 180.00000} ; insert
  LIN {X -13926.877,Y 2173.194,Z -151.962,A -45.04237,B 0.00000,C 180.00000} ; release
  LIN {X -13926.877,Y 2173.194,Z 148.038,A -45.04237,B 0.00000,C 180.00000} ; retreat
  ; Step 421, bar 3132
  LIN {X -14073.123,Y 2173.194,Z 947.644,A -134.95763,B 0.00000,C -180.00000} ; outside
  LIN {X -14073.123,Y 2173.194,Z 98.038,A -134.95763,B 0.00000,C -180.00000} ; preinsert
  LIN {X -14073.123,Y 2173.194,Z -151.962,A -134.95763,B 0.00000,C -180.00000} ; insert
  LIN {X -14073.123,Y 2173.194,Z -151.962,A -134.95763,B 0.00000,C -180.00000} ; release
  LIN {X -14073.123,Y 2173.194,Z 148.038,A -134.95763,B 0.00000,C -180.00000} ; retreat
  ; Step 422, bar 1241
  LIN {X -13149.921,Y 0.110,Z 819.136,A 89.99666,B 0.00000,C 180.00000} ; outside
  LIN {X -13149.921,Y 0.110,Z -29.671,A 89.99666,B 0.00000,C 180.00000} ; preinsert
  LIN {X -13149.921,Y 0.110,Z -279.671,A 89.99666,B 0.00000,C 180.00000} ; insert
  LIN {X -13149.921,Y 0.110,Z -279.671,A 89.99666,B 0.00000,C 180.00000} ; release
  LIN {X -13149.921,Y 0.110,Z 20.329,A 89.99666,B 0.00000,C 180.00000} ; retreat
  ; Step 423, bar 1026
  LIN {X 13149.921,Y 0.097,Z 819.136,A 90.00334,B 0.00000,C 180.00000} ; outside
  LIN {X 13149.921,Y 0.097,Z -29.671,A 90.00334,B 0.00000,C 180.00000} ; preinsert
  LIN {X 13149.921,Y 0.097,Z -279.671,A 90.00334,B 0.00000,C 180.00000} ; insert
  LIN {X 13149.921,Y 0.097,Z -279.671,A 90.00334,B 0.00000,C 180.00000} ; release
  LIN {X 13149.921,Y 0.097,Z 20.329,A 90.00334,B 0.00000,C 180.00000} ; retreat
  ; Step 424, bar 1240
  LIN {X -13049.921,Y 0.110,Z 832.498,A 89.99666,B 0.00000,C 180.00000} ; outside
  LIN {X -13049.921,Y 0.110,Z -22.991,A 89.99666,B 0.00000,C 180.00000} ; preinsert
  LIN {X -13049.921,Y 0.110,Z -272.991,A 89.99666,B 0.00000,C 180.00000} ; insert
  LIN {X -13049.921,Y 0.110,Z -272.991,A 89.99666,B 0.00000,C 180.00000} ; release
  LIN {X -13049.921,Y 0.110,Z 27.009,A 89.99666,B 0.00000,C 180.00000} ; retreat
  ; Step 425, bar 1025
  LIN {X 13049.921,Y 0.097,Z 832.498,A 90.00334,B 0.00000,C 180.00000} ; outside
  LIN {X 13049.921,Y 0.097,Z -22.991,A 90.00334,B 0.00000,C 180.00000} ; preinsert
  LIN {X 13049.921,Y 0.097,Z -272.991,A 90.00334,B 0.00000,C 180.00000} ; insert
  LIN {X 13049.921,Y 0.097,Z -272.991,A 90.00334,B 0.00000,C 180.00000} ; release
  LIN {X 13049.921,Y 0.097,Z 27.009,A 90.00334,B 0.00000,C 180.00000} ; retreat
  ; Step 426, bar 1239
  LIN {X -12949.921,Y 0.110,Z 845.860,A 89.99666,B 0.00000,C 180.00000} ; outside
  LIN {X -12949.921,Y 0.110,Z -16.310,A 89.99666,B 0.00000,C 180.00000} ; preinsert
  LIN {X -12949.921,Y 0.110,Z -266.310,A 89.99666,B 0.00000,C 180.00000} ; insert
  LIN {X -12949.921,Y 0.110,Z -266.310,A 89.99666,B 0.00000,C 180.00000} ; release
  LIN {X -12949.921,Y 0.110,Z 33.690,A 89.99666,B 0.00000,C 180.00000} ; retreat
  ; Step 427, bar 1024
  LIN {X 12949.921,Y 0.097,Z 845.860,A 90.00334,B 0.00000,C 180.00000} ; outside
  LIN {X 12949.921,Y 0.097,Z -16.310,A 90.00334,B 0.00000,C 180.00000} ; preinsert
  LIN {X 12949.921,Y 0.097,Z -266.310,A 90.00334,B 0.00000,C 180.00000} ; insert
  LIN {X 12949.921,Y 0.097,Z -266.310,A 90.00334,B 0.00000,C 180.00000} ; release
  LIN {X 12949.921,Y 0.097,Z 33.690,A 90.00334,B 0.00000,C 180.00000} ; retreat
  ; Step 428, bar 1248
  LIN {X -12865.921,Y 0.110,Z 859.221,A 89.99666,B 0.00000,C 180.00000} ; outside
  LIN {X -12865.921,Y 0.110,Z -9.629,A 89.99666,B 0.00000,C 180.00000} ; preinsert
  LIN {X -12865.921,Y 0.110,Z -259.629,A 89.99666,B 0.00000,C 180.00000} ; insert
  LIN {X -12865.921,Y 0.110,Z -259.629,A 89.99666,B 0.00000,C 180.00000} ; release
  LIN {X -12865.921,Y 0.110,Z 40.371,A 89.99666,B 0.00000,C 180.00000} ; retreat
  ; Step 429, bar 1238
  LIN {X -12849.921,Y 0.110,Z 859.221,A 89.99666,B 0.00000,C 180.00000} ; outside
  LIN {X -12849.921,Y 0.110,Z -9.629,A 89.99666,B 0.00000,C 180.00000} ; preinsert
  LIN {X -12849.921,Y 0.110,Z -259.629,A 89.99666,B 0.00000,C 180.00000} ; insert
  LIN {X -12849.921,Y 0.110,Z -259.629,A 89.99666,B 0.00000,C 180.00000} ; release
  LIN {X -12849.921,Y 0.110,Z 40.371,A 89.99666,B 0.00000,C 180.00000} ; retreat
  ; Step 430, bar 1023
  LIN {X 12849.921,Y 0.097,Z 859.221,A 90.00334,B 0.00000,C 180.00000} ; outside
  LIN {X 12849.921,Y 0.097,Z -9.629,A 90.00334,B 0.00000,C 180.00000} ; preinsert
  LIN {X 12849.921,Y 0.097,Z -259.629,A 90.00334,B 0.00000,C 180.00000} ; insert
  LIN {X 12849.921,Y 0.097,Z -259.629,A 90.00334,B 0.00000,C 180.00000} ; release
  LIN {X 12849.921,Y 0.097,Z 40.371,A 90.00334,B 0.00000,C 180.00000} ; retreat
  ; Step 431, bar 1034
  LIN {X 12865.921,Y 0.097,Z 859.221,A 90.00334,B 0.00000,C 180.00000} ; outside
  LIN {X 12865.921,Y 0.097,Z -9.629,A 90.00334,B 0.00000,C 180.00000} ; preinsert
  LIN {X 12865.921,Y 0.097,Z -259.629,A 90.00334,B 0.00000,C 180.00000} ; insert
  LIN {X 12865.921,Y 0.097,Z -259.629,A 90.00334,B 0.00000,C 180.00000} ; release
  LIN {X 12865.921,Y 0.097,Z 40.371,A 90.00334,B 0.00000,C 180.00000} ; retreat
  ; Step 432, bar 1237
  LIN {X -12749.921,Y 0.110,Z 872.583,A 89.99666,B 0.00000,C 180.00000} ; outside
  LIN {X -12749.921,Y 0.110,Z -2.948,A 89.99666,B 0.00000,C 180.00000} ; preinsert
  LIN {X -12749.921,Y 0.110,Z -252.948,A 89.99666,B 0.00000,C 180.00000} ; insert
  LIN {X -12749.921,Y 0.110,Z -252.948,A 89.99666,B 0.00000,C 180.00000} ; release
  LIN {X -12749.921,Y 0.110,Z 47.052,A 89.99666,B 0.00000,C 180.00000} ; retreat
  ; Step 433, bar 1022
  LIN {X 12749.921,Y 0.097,Z 872.583,A 90.00334,B 0.00000,C 180.00000} ; outside
  LIN {X 12749.921,Y 0.097,Z -2.948,A 90.00334,B 0.00000,C 180.00000} ; preinsert
  LIN {X 12749.921,Y 0.097,Z -252.948,A 90.00334,B 0.00000,C 180.00000} ; insert
  LIN {X 12749.921,Y 0.097,Z -252.948,A 90.00334,B 0.00000,C 180.00000} ; release
  LIN {X 12749.921,Y 0.097,Z 47.052,A 90.00334,B 0.00000,C 180.00000} ; retreat
  ; Step 434, bar 1236
  LIN {X -12649.921,Y 0.110,Z 885.945,A 89.99666,B 0.00000,C 180.00000} ; outside
  LIN {X -12649.921,Y 0.110,Z 3.733,A 89.99666,B 0.00000,C 180.00000} ; preinsert
  LIN {X -12649.921,Y 0.110,Z -246.267,A 89.99666,B 0.00000,C 180.00000} ; insert
  LIN {X -12649.921,Y 0.110,Z -246.267,A 89.99666,B 0.00000,C 180.00000} ; release
  LIN {X -12649.921,Y 0.110,Z 53.733,A 89.99666,B 0.00000,C 180.00000} ; retreat
  ; Step 435, bar 1021
  LIN {X 12649.921,Y 0.097,Z 885.945,A 90.00334,B 0.00000,C 180.00000} ; outside
  LIN {X 12649.921,Y 0.097,Z 3.733,A 90.00334,B 0.00000,C 180.00000} ; preinsert
  LIN {X 12649.921,Y 0.097,Z -246.267,A 90.00334,B 0.00000,C 180.00000} ; insert
  LIN {X 12649.921,Y 0.097,Z -246.267,A 90.00334,B 0.00000,C 180.00000} ; release
  LIN {X 12649.921,Y 0.097,Z 53.733,A 90.00334,B 0.00000,C 180.00000} ; retreat
  ; Step 436, bar 1235
  LIN {X -12549.921,Y 0.110,Z 899.306,A 89.99666,B 0.00000,C 180.00000} ; outside
  LIN {X -12549.921,Y 0.110,Z 10.414,A 89.99666,B 0.00000,C 180.00000} ; preinsert
  LIN {X -12549.921,Y 0.110,Z -239.586,A 89.99666,B 0.00000,C 180.00000} ; insert
  LIN {X -12549.921,Y 0.110,Z -239.586,A 89.99666,B 0.00000,C 180.00000} ; release
  LIN {X -12549.921,Y 0.110,Z 60.414,A 89.99666,B 0.00000,C 180.00000} ; retreat
  ; Step 437, bar 1020
  LIN {X 12549.921,Y 0.097,Z 899.306,A 90.00334,B 0.00000,C 180.00000} ; outside
  LIN {X 12549.921,Y 0.097,Z 10.414,A 90.00334,B 0.00000,C 180.00000} ; preinsert
  LIN {X 12549.921,Y 0.097,Z -239.586,A 90.00334,B 0.00000,C 180.00000} ; insert
  LIN {X 12549.921,Y 0.097,Z -239.586,A 90.00334,B 0.00000,C 180.00000} ; release
  LIN {X 12549.921,Y 0.097,Z 60.414,A 90.00334,B 0.00000,C 180.00000} ; retreat
  ; Step 438, bar 297
  LIN {X 0.000,Y -2590.000,Z 1034.371,A 0.00000,B 0.00000,C 180.00000} ; outside
  LIN {X 0.000,Y -2590.000,Z 141.496,A 0.00000,B 0.00000,C 180.00000} ; preinsert
  LIN {X 0.000,Y -2590.000,Z -108.504,A 0.00000,B 0.00000,C 180.00000} ; insert
  LIN {X 0.000,Y -2590.000,Z -108.504,A 0.00000,B 0.00000,C 180.00000} ; release
  LIN {X 0.000,Y -2590.000,Z 191.496,A 0.00000,B 0.00000,C 180.00000} ; retreat
  ; Step 439, bar 324
  LIN {X 0.000,Y 2590.000,Z 1034.371,A 0.00000,B 0.00000,C 180.00000} ; outside
  LIN {X 0.000,Y 2590.000,Z 141.496,A 0.00000,B 0.00000,C 180.00000} ; preinsert
  LIN {X 0.000,Y 2590.000,Z -108.504,A 0.00000,B 0.00000,C 180.00000} ; insert
  LIN {X 0.000,Y 2590.000,Z -108.504,A 0.00000,B 0.00000,C 180.00000} ; release
  LIN {X 0.000,Y 2590.000,Z 191.496,A 0.00000,B 0.00000,C 180.00000} ; retreat
  ; Step 440, bar 1919
  LIN {X -15076.912,Y -2150.800,Z 792.677,A -179.99743,B 0.00000,C 180.00000} ; outside
  LIN {X -15076.912,Y -2150.800,Z -105.163,A -179.99743,B 0.00000,C 180.00000} ; preinsert
  LIN {X -15076.912,Y -2150.800,Z -355.163,A -179.99743,B 0.00000,C 180.00000} ; insert
  LIN {X -15076.912,Y -2150.800,Z -355.163,A -179.99743,B 0.00000,C 180.00000} ; release
  LIN {X -15076.912,Y -2150.800,Z -55.163,A -179.99743,B 0.00000,C 180.00000} ; retreat
  ; Step 441, bar 1903
  LIN {X 15076.912,Y -2150.800,Z 792.677,A -0.00257,B 0.00000,C 180.00000} ; outside
  LIN {X 15076.912,Y -2150.800,Z -105.163,A -0.00257,B 0.00000,C 180.00000} ; preinsert
  LIN {X 15076.912,Y -2150.800,Z -355.163,A -0.00257,B 0.00000,C 180.00000} ; insert
  LIN {X 15076.912,Y -2150.800,Z -355.163,A -0.00257,B 0.00000,C 180.00000} ; release
  LIN {X 15076.912,Y -2150.800,Z -55.163,A -0.00257,B 0.00000,C 180.00000} ; retreat
  ; Step 442, bar 1920
  LIN {X -15076.912,Y 2150.800,Z 792.677,A 179.99743,B 0.00000,C -180.00000} ; outside
  LIN {X -15076.912,Y 2150.800,Z -105.163,A 179.99743,B 0.00000,C -180.00000} ; preinsert
  LIN {X -15076.912,Y 2150.800,Z -355.163,A 179.99743,B 0.00000,C -180.00000} ; insert
  LIN {X -15076.912,Y 2150.800,Z -355.163,A 179.99743,B 0.00000,C -180.00000} ; release
  LIN {X -15076.912,Y 2150.800,Z -55.163,A 179.99743,B 0.00000,C -180.00000} ; retreat
  ; Step 443, bar 1904
  LIN {X 15076.912,Y 2150.800,Z 792.677,A 0.00257,B 0.00000,C 180.00000} ; outside
  LIN {X 15076.912,Y 2150.800,Z -105.163,A 0.00257,B 0.00000,C 180.00000} ; preinsert
  LIN {X 15076.912,Y 2150.800,Z -355.163,A 0.00257,B 0.00000,C 180.00000} ; insert
  LIN {X 15076.912,Y 2150.800,Z -355.163,A 0.00257,B 0.00000,C 180.00000} ; release
  LIN {X 15076.912,Y 2150.800,Z -55.163,A 0.00257,B 0.00000,C 180.00000} ; retreat
  ; Step 444, bar 296
  LIN {X 0.000,Y -2455.000,Z 1040.621,A 0.00000,B 0.00000,C 180.00000} ; outside
  LIN {X 0.000,Y -2455.000,Z 144.621,A 0.00000,B 0.00000,C 180.00000} ; preinsert
  LIN {X 0.000,Y -2455.000,Z -105.379,A 0.00000,B 0.00000,C 180.00000} ; insert
  LIN {X 0.000,Y -2455.000,Z -105.379,A 0.00000,B 0.00000,C 180.00000} ; release
  LIN {X 0.000,Y -2455.000,Z 194.621,A 0.00000,B 0.00000,C 180.00000} ; retreat
  ; Step 445, bar 323
  LIN {X 0.000,Y 2455.000,Z 1040.621,A 0.00000,B 0.00000,C 180.00000} ; outside
  LIN {X 0.000,Y 2455.000,Z 144.621,A 0.00000,B 0.00000,C 180.00000} ; preinsert
  LIN {X 0.000,Y 2455.000,Z -105.379,A 0.00000,B 0.00000,C 180.00000} ; insert
  LIN {X 0.000,Y 2455.000,Z -105.379,A 0.00000,B 0.00000,C 180.00000} ; release
  LIN {X 0.000,Y 2455.000,Z 194.621,A 0.00000,B 0.00000,C 180.00000} ; retreat
  ; Step 446, bar 1247
  LIN {X -12465.921,Y 0.110,Z 912.668,A 89.99666,B 0.00000,C 180.00000} ; outside
  LIN {X -12465.921,Y 0.110,Z 17.094,A 89.99666,B 0.00000,C 180.00000} ; preinsert
  LIN {X -12465.921,Y 0.110,Z -232.906,A 89.99666,B 0.00000,C 180.00000} ; insert
  LIN {X -12465.921,Y 0.110,Z -232.906,A 89.99666,B 0.00000,C 180.00000} ; release
  LIN {X -12465.921,Y 0.110,Z 67.094,A 89.99666,B 0.00000,C 180.00000} ; retreat
  ; Step 447, bar 1234
  LIN {X -12449.921,Y 0.110,Z 912.668,A 89.99666,B 0.00000,C 180.00000} ; outside
  LIN {X -12449.921,Y 0.110,Z 17.094,A 89.99666,B 0.00000,C 180.00000} ; preinsert
  LIN {X -12449.921,Y 0.110,Z -232.906,A 89.99666,B 0.00000,C 180.00000} ; insert
  LIN {X -12449.921,Y 0.110,Z -232.906,A 89.99666,B 0.00000,C 180.00000} ; release
  LIN {X -12449.921,Y 0.110,Z 67.094,A 89.99666,B 0.00000,C 180.00000} ; retreat
  ; Step 448, bar 1019
  LIN {X 12449.921,Y 0.097,Z 912.668,A 90.00334,B 0.00000,C 180.00000} ; outside
  LIN {X 12449.921,Y 0.097,Z 17.094,A 90.00334,B 0.00000,C 180.00000} ; preinsert
  LIN {X 12449.921,Y 0.097,Z -232.906,A 90.00334,B 0.00000,C 180.00000} ; insert
  LIN {X 12449.921,Y 0.097,Z -232.906,A 90.00334,B 0.00000,C 180.00000} ; release
